LIN {X 0,Y 412.473,Z 356.373,A -85,B 0,C 180,E1 -10488.564,E2 -10488.564} C_VEL
LIN {X 0,Y 413.855,Z 363.338,A -85,B 0,C 180,E1 -10491.872,E2 -10491.872} C_VEL
LIN {X 0,Y 414.561,Z 368.323,A -85,B 0,C 180,E1 -10494.091,E2 -10494.091} C_VEL
LIN {X 0,Y 414.047,Z 374.671,A -85,B 0,C 180,E1 -10496.674,E2 -10496.674} C_VEL
LIN {X 0,Y 413.079,Z 384.313,A -85,B 0,C 180,E1 -10500.435,E2 -10500.435} C_VEL
LIN {X 0,Y 412.15,Z 394.191,A -85,B 0,C 180,E1 -10504.226,E2 -10504.226} C_VEL
LIN {X 0,Y 411.927,Z 397.665,A -85,B 0,C 180,E1 -10505.56,E2 -10505.56} C_VEL
LIN {X 0,Y 415.986,Z 414.745,A -85,B 0,C 180,E1 -10506.23,E2 -10506.23} C_VEL
LIN {X 0,Y 418.674,Z 429.42,A -85,B 0,C 180,E1 -10506.952,E2 -10506.952} C_VEL
LIN {X 0,Y 419.189,Z 434.682,A -85,B 0,C 180,E1 -10507.237,E2 -10507.237} C_VEL
LIN {X 0,Y 418.226,Z 448.445,A -85,B 0,C 180,E1 -10507.985,E2 -10507.985} C_VEL
LIN {X 0,Y 417.116,Z 461.685,A -85,B 0,C 180,E1 -10508.89,E2 -10508.89} C_VEL
LIN {X 0,Y 415.821,Z 474.731,A -85,B 0,C 180,E1 -10509.985,E2 -10509.985} C_VEL
LIN {X 0,Y 414.639,Z 486.804,A -85,B 0,C 180,E1 -10511.213,E2 -10511.213} C_VEL
LIN {X 0,Y 413.542,Z 498.914,A -85,B 0,C 180,E1 -10512.698,E2 -10512.698} C_VEL
LIN {X 0,Y 412.48,Z 509.113,A -85,B 0,C 180,E1 -10514.18,E2 -10514.18} C_VEL
LIN {X 0,Y 411.633,Z 519.099,A -85,B 0,C 180,E1 -10515.919,E2 -10515.919} C_VEL
LIN {X 0,Y 410.992,Z 527.441,A -85,B 0,C 180,E1 -10517.658,E2 -10517.658} C_VEL
LIN {X 0,Y 410.621,Z 533.414,A -85,B 0,C 180,E1 -10519.148,E2 -10519.148} C_VEL
LIN {X 0,Y 410.225,Z 539.99,A -85,B 0,C 180,E1 -10521.13,E2 -10521.13} C_VEL
LIN {X 0,Y 410.058,Z 545.099,A -85,B 0,C 180,E1 -10523.109,E2 -10523.109} C_VEL
LIN {X 0,Y 409.992,Z 548.857,A -85,B 0,C 180,E1 -10525.083,E2 -10525.083} C_VEL
LIN {X 0,Y 409.971,Z 551.337,A -85,B 0,C 180,E1 -10527.052,E2 -10527.052} C_VEL
LIN {X 0,Y 409.974,Z 552.586,A -85,B 0,C 180,E1 -10529.018,E2 -10529.018} C_VEL
LIN {X 0,Y 409.974,Z 552.585,A -85,B 0,C 180,E1 -10530.982,E2 -10530.982} C_VEL
LIN {X 0,Y 409.971,Z 551.33,A -85,B 0,C 180,E1 -10532.948,E2 -10532.948} C_VEL
LIN {X 0,Y 409.998,Z 548.848,A -85,B 0,C 180,E1 -10534.917,E2 -10534.917} C_VEL
LIN {X 0,Y 410.068,Z 545.095,A -85,B 0,C 180,E1 -10536.89,E2 -10536.89} C_VEL
LIN {X 0,Y 410.225,Z 539.984,A -85,B 0,C 180,E1 -10538.87,E2 -10538.87} C_VEL
LIN {X 0,Y 410.621,Z 533.397,A -85,B 0,C 180,E1 -10540.852,E2 -10540.852} C_VEL
LIN {X 0,Y 411.011,Z 526.298,A -85,B 0,C 180,E1 -10542.593,E2 -10542.593} C_VEL
LIN {X 0,Y 411.745,Z 517.767,A -85,B 0,C 180,E1 -10544.33,E2 -10544.33} C_VEL
LIN {X 0,Y 412.642,Z 507.498,A -85,B 0,C 180,E1 -10546.067,E2 -10546.067} C_VEL
LIN {X 0,Y 413.651,Z 497.039,A -85,B 0,C 180,E1 -10547.552,E2 -10547.552} C_VEL
LIN {X 0,Y 414.933,Z 484.534,A -85,B 0,C 180,E1 -10549.029,E2 -10549.029} C_VEL
LIN {X 0,Y 416.072,Z 472.024,A -85,B 0,C 180,E1 -10550.26,E2 -10550.26} C_VEL
LIN {X 0,Y 417.353,Z 458.355,A -85,B 0,C 180,E1 -10551.356,E2 -10551.356} C_VEL
LIN {X 0,Y 418.476,Z 445.087,A -85,B 0,C 180,E1 -10552.215,E2 -10552.215} C_VEL
LIN {X 0,Y 419.176,Z 432.684,A -85,B 0,C 180,E1 -10552.861,E2 -10552.861} C_VEL
LIN {X 0,Y 416.901,Z 419.271,A -85,B 0,C 180,E1 -10553.554,E2 -10553.554} C_VEL
LIN {X 0,Y 413.581,Z 404.549,A -85,B 0,C 180,E1 -10554.182,E2 -10554.182} C_VEL
LIN {X 0,Y 411.925,Z 397.627,A -85,B 0,C 180,E1 -10554.44,E2 -10554.44} C_VEL
LIN {X 0,Y 412.667,Z 388.34,A -85,B 0,C 180,E1 -10558.01,E2 -10558.01} C_VEL
LIN {X 0,Y 413.477,Z 380.023,A -85,B 0,C 180,E1 -10561.226,E2 -10561.226} C_VEL
LIN {X 0,Y 414.356,Z 371.385,A -85,B 0,C 180,E1 -10564.625,E2 -10564.625} C_VEL
LIN {X 0,Y 414.582,Z 368.286,A -85,B 0,C 180,E1 -10565.908,E2 -10565.908} C_VEL
LIN {X 0,Y 413.649,Z 362.257,A -85,B 0,C 180,E1 -10568.597,E2 -10568.597} C_VEL
LIN {X 0,Y 412.154,Z 354.701,A -85,B 0,C 180,E1 -10572.237,E2 -10572.237} C_VEL
LIN {X 0,Y 411.206,Z 349.895,A -85,B 0,C 180,E1 -10574.733,E2 -10574.733} C_VEL
LIN {X 0,Y 411.2,Z 349.883,A -85,B 0,C 180,E1 -10578.198,E2 -10578.198} C_VEL
LIN {X 0,Y 411.234,Z 349.887,A -85,B 0,C 180,E1 -10580.778,E2 -10580.778} C_VEL
LIN {X 0,Y 411.202,Z 349.895,A -85,B 0,C 180,E1 -10584.472,E2 -10584.472} C_VEL
LIN {X 0,Y 411.209,Z 349.892,A -85,B 0,C 180,E1 -10586.874,E2 -10586.874} C_VEL
LIN {X 0,Y 411.235,Z 349.886,A -85,B 0,C 180,E1 -10590.644,E2 -10590.644} C_VEL
LIN {X 0,Y 411.241,Z 349.885,A -85,B 0,C 180,E1 -10593.619,E2 -10593.619} C_VEL
LIN {X 0,Y 411.207,Z 349.888,A -85,B 0,C 180,E1 -10596.853,E2 -10596.853} C_VEL
LIN {X 0,Y 411.219,Z 349.887,A -85,B 0,C 180,E1 -10600.05,E2 -10600.05} C_VEL
LIN {X 0,Y 411.266,Z 349.881,A -85,B 0,C 180,E1 -10603.131,E2 -10603.131} C_VEL
LIN {X 0,Y 411.317,Z 349.87,A -85,B 0,C 180,E1 -10606.891,E2 -10606.891} C_VEL
LIN {X 0,Y 411.298,Z 349.874,A -85,B 0,C 180,E1 -10610.162,E2 -10610.162} C_VEL
LIN {X 0,Y 411.447,Z 349.857,A -85,B 0,C 180,E1 -10613.133,E2 -10613.133} C_VEL
LIN {X 0,Y 411.313,Z 349.877,A -85,B 0,C 180,E1 -10615.099,E2 -10615.099} C_VEL
LIN {X 0,Y 411.516,Z 349.849,A -85,B 0,C 180,E1 -10618.043,E2 -10618.043} C_VEL
LIN {X 0,Y 411.645,Z 349.831,A -85,B 0,C 180,E1 -10620,E2 -10620} C_VEL
LIN {X 0,Y 411.461,Z 349.858,A -85,B 0,C 180,E1 -10622.937,E2 -10622.937} C_VEL
LIN {X 0,Y 411.465,Z 349.855,A -85,B 0,C 180,E1 -10626.867,E2 -10626.867} C_VEL
LIN {X 0,Y 411.311,Z 349.878,A -85,B 0,C 180,E1 -10629.838,E2 -10629.838} C_VEL
LIN {X 0,Y 411.318,Z 349.876,A -85,B 0,C 180,E1 -10633.109,E2 -10633.109} C_VEL
LIN {X 0,Y 411.261,Z 349.882,A -85,B 0,C 180,E1 -10636.889,E2 -10636.889} C_VEL
LIN {X 0,Y 411.234,Z 349.888,A -85,B 0,C 180,E1 -10639.987,E2 -10639.987} C_VEL
LIN {X 0,Y 411.207,Z 349.89,A -85,B 0,C 180,E1 -10643.147,E2 -10643.147} C_VEL
LIN {X 0,Y 411.242,Z 349.884,A -85,B 0,C 180,E1 -10646.381,E2 -10646.381} C_VEL
LIN {X 0,Y 411.204,Z 349.886,A -85,B 0,C 180,E1 -10649.713,E2 -10649.713} C_VEL
LIN {X 0,Y 411.21,Z 349.888,A -85,B 0,C 180,E1 -10653.156,E2 -10653.156} C_VEL
LIN {X 0,Y 411.196,Z 349.891,A -85,B 0,C 180,E1 -10656.553,E2 -10656.553} C_VEL
LIN {X 0,Y 411.216,Z 349.889,A -85,B 0,C 180,E1 -10659.728,E2 -10659.728} C_VEL
LIN {X 0,Y 411.177,Z 349.893,A -85,B 0,C 180,E1 -10663.133,E2 -10663.133} C_VEL
LIN {X 0,Y 411.171,Z 349.896,A -85,B 0,C 180,E1 -10665.881,E2 -10665.881} C_VEL
LIN {X 0,Y 411.242,Z 350.049,A -85,B 0,C 180,E1 -10667.531,E2 -10667.531} C_VEL
LIN {X 0,Y 411.73,Z 353.5,A -85,B 0,C 180,E1 -10670.186,E2 -10670.186} C_VEL
LIN {X 0,Y 411.809,Z 356.083,A -85,B 0,C 180,E1 -10672.093,E2 -10672.093} C_VEL
LIN {X 0,Y 411.664,Z 360.213,A -85,B 0,C 180,E1 -10675.032,E2 -10675.032} C_VEL
LIN {X 0,Y 411.374,Z 364.529,A -85,B 0,C 180,E1 -10678.021,E2 -10678.021} C_VEL
LIN {X 0,Y 411.101,Z 369.543,A -85,B 0,C 180,E1 -10681.401,E2 -10681.401} C_VEL
LIN {X 0,Y 410.923,Z 374.622,A -85,B 0,C 180,E1 -10684.686,E2 -10684.686} C_VEL
LIN {X 0,Y 410.712,Z 380.389,A -85,B 0,C 180,E1 -10688.235,E2 -10688.235} C_VEL
LIN {X 0,Y 415.732,Z 397.121,A -85,B 0,C 180,E1 -10688.991,E2 -10688.991} C_VEL
LIN {X 0,Y 418.903,Z 410.203,A -85,B 0,C 180,E1 -10689.72,E2 -10689.72} C_VEL
LIN {X 0,Y 418.637,Z 418.558,A -85,B 0,C 180,E1 -10690.151,E2 -10690.151} C_VEL
LIN {X 0,Y 417.778,Z 431.637,A -85,B 0,C 180,E1 -10690.978,E2 -10690.978} C_VEL
LIN {X 0,Y 416.805,Z 443.798,A -85,B 0,C 180,E1 -10691.951,E2 -10691.951} C_VEL
LIN {X 0,Y 415.674,Z 454.932,A -85,B 0,C 180,E1 -10693.043,E2 -10693.043} C_VEL
LIN {X 0,Y 414.628,Z 465.155,A -85,B 0,C 180,E1 -10694.264,E2 -10694.264} C_VEL
LIN {X 0,Y 413.718,Z 473.99,A -85,B 0,C 180,E1 -10695.532,E2 -10695.532} C_VEL
LIN {X 0,Y 412.839,Z 482.36,A -85,B 0,C 180,E1 -10696.964,E2 -10696.964} C_VEL
LIN {X 0,Y 411.999,Z 489.544,A -85,B 0,C 180,E1 -10698.438,E2 -10698.438} C_VEL
LIN {X 0,Y 411.306,Z 496.408,A -85,B 0,C 180,E1 -10700.162,E2 -10700.162} C_VEL
LIN {X 0,Y 410.725,Z 502.566,A -85,B 0,C 180,E1 -10702.132,E2 -10702.132} C_VEL
LIN {X 0,Y 410.437,Z 507.144,A -85,B 0,C 180,E1 -10704.103,E2 -10704.103} C_VEL
LIN {X 0,Y 410.166,Z 510.317,A -85,B 0,C 180,E1 -10706.07,E2 -10706.07} C_VEL
LIN {X 0,Y 410.071,Z 512.187,A -85,B 0,C 180,E1 -10708.036,E2 -10708.036} C_VEL
LIN {X 0,Y 409.971,Z 512.826,A -85,B 0,C 180,E1 -10710,E2 -10710} C_VEL
LIN {X 0,Y 410.07,Z 512.25,A -85,B 0,C 180,E1 -10711.964,E2 -10711.964} C_VEL
LIN {X 0,Y 410.164,Z 510.414,A -85,B 0,C 180,E1 -10713.954,E2 -10713.954} C_VEL
LIN {X 0,Y 410.432,Z 507.339,A -85,B 0,C 180,E1 -10715.897,E2 -10715.897} C_VEL
LIN {X 0,Y 410.722,Z 502.824,A -85,B 0,C 180,E1 -10717.868,E2 -10717.868} C_VEL
LIN {X 0,Y 410.764,Z 502.241,A -85,B 0,C 180,E1 -10718.078,E2 -10718.078} C_VEL
LIN {X 0,Y 410.259,Z 500.112,A -85,B 0,C 180,E1 -10718.844,E2 -10718.844} C_VEL
LIN {X 0,Y 407.69,Z 496.379,A -85,B 0,C 180,E1 -10720.086,E2 -10720.086} C_VEL
LIN {X 0,Y 405.311,Z 492.191,A -85,B 0,C 180,E1 -10721.307,E2 -10721.307} C_VEL
LIN {X 0,Y 405.102,Z 489.194,A -85,B 0,C 180,E1 -10722.029,E2 -10722.029} C_VEL
LIN {X 0,Y 406.031,Z 481.921,A -85,B 0,C 180,E1 -10723.514,E2 -10723.514} C_VEL
LIN {X 0,Y 406.961,Z 473.123,A -85,B 0,C 180,E1 -10725.013,E2 -10725.013} C_VEL
LIN {X 0,Y 407.969,Z 464.366,A -85,B 0,C 180,E1 -10726.257,E2 -10726.257} C_VEL
LIN {X 0,Y 409.145,Z 452.742,A -85,B 0,C 180,E1 -10727.623,E2 -10727.623} C_VEL
LIN {X 0,Y 410.309,Z 441.068,A -85,B 0,C 180,E1 -10728.733,E2 -10728.733} C_VEL
LIN {X 0,Y 411.399,Z 428.167,A -85,B 0,C 180,E1 -10729.718,E2 -10729.718} C_VEL
LIN {X 0,Y 412.277,Z 415.028,A -85,B 0,C 180,E1 -10730.501,E2 -10730.501} C_VEL
LIN {X 0,Y 412.268,Z 411.549,A -85,B 0,C 180,E1 -10730.687,E2 -10730.687} C_VEL
LIN {X 0,Y 409.079,Z 398.314,A -85,B 0,C 180,E1 -10731.455,E2 -10731.455} C_VEL
LIN {X 0,Y 404.658,Z 383.818,A -85,B 0,C 180,E1 -10732.15,E2 -10732.15} C_VEL
LIN {X 0,Y 403.732,Z 380.544,A -85,B 0,C 180,E1 -10732.295,E2 -10732.295} C_VEL
LIN {X 0,Y 403.891,Z 374.995,A -85,B 0,C 180,E1 -10735.787,E2 -10735.787} C_VEL
LIN {X 0,Y 404.125,Z 369.877,A -85,B 0,C 180,E1 -10739.14,E2 -10739.14} C_VEL
LIN {X 0,Y 404.396,Z 364.864,A -85,B 0,C 180,E1 -10742.599,E2 -10742.599} C_VEL
LIN {X 0,Y 404.7,Z 359.772,A -85,B 0,C 180,E1 -10746.189,E2 -10746.189} C_VEL
LIN {X 0,Y 404.856,Z 356.353,A -85,B 0,C 180,E1 -10748.678,E2 -10748.678} C_VEL
LIN {X 0,Y 404.475,Z 352.452,A -85,B 0,C 180,E1 -10751.656,E2 -10751.656} C_VEL
LIN {X 0,Y 404.18,Z 350.766,A -85,B 0,C 180,E1 -10753.087,E2 -10753.087} C_VEL
LIN {X 0,Y 404.157,Z 350.765,A -85,B 0,C 180,E1 -10756.916,E2 -10756.916} C_VEL
LIN {X 0,Y 404.173,Z 350.763,A -85,B 0,C 180,E1 -10759.956,E2 -10759.956} C_VEL
LIN {X 0,Y 404.141,Z 350.77,A -85,B 0,C 180,E1 -10763.125,E2 -10763.125} C_VEL
LIN {X 0,Y 404.149,Z 350.767,A -85,B 0,C 180,E1 -10766.188,E2 -10766.188} C_VEL
LIN {X 0,Y 404.15,Z 350.768,A -85,B 0,C 180,E1 -10769.715,E2 -10769.715} C_VEL
LIN {X 0,Y 404.201,Z 350.764,A -85,B 0,C 180,E1 -10773.123,E2 -10773.123} C_VEL
LIN {X 0,Y 404.182,Z 350.764,A -85,B 0,C 180,E1 -10775.334,E2 -10775.334} C_VEL
LIN {X 0,Y 404.144,Z 350.766,A -85,B 0,C 180,E1 -10778.581,E2 -10778.581} C_VEL
LIN {X 0,Y 404.214,Z 350.758,A -85,B 0,C 180,E1 -10781.762,E2 -10781.762} C_VEL
LIN {X 0,Y 404.212,Z 350.758,A -85,B 0,C 180,E1 -10784.882,E2 -10784.882} C_VEL
LIN {X 0,Y 404.262,Z 350.752,A -85,B 0,C 180,E1 -10787.958,E2 -10787.958} C_VEL
LIN {X 0,Y 404.439,Z 350.732,A -85,B 0,C 180,E1 -10792.099,E2 -10792.099} C_VEL
LIN {X 0,Y 404.43,Z 350.73,A -85,B 0,C 180,E1 -10794.015,E2 -10794.015} C_VEL
LIN {X 0,Y 404.486,Z 350.723,A -85,B 0,C 180,E1 -10798.008,E2 -10798.008} C_VEL
LIN {X 0,Y 404.615,Z 350.712,A -85,B 0,C 180,E1 -10800,E2 -10800} C_VEL
LIN {X 0,Y 404.42,Z 350.733,A -85,B 0,C 180,E1 -10802.988,E2 -10802.988} C_VEL
LIN {X 0,Y 404.419,Z 350.733,A -85,B 0,C 180,E1 -10805.985,E2 -10805.985} C_VEL
LIN {X 0,Y 404.272,Z 350.754,A -85,B 0,C 180,E1 -10809.001,E2 -10809.001} C_VEL
LIN {X 0,Y 404.274,Z 350.756,A -85,B 0,C 180,E1 -10812.041,E2 -10812.041} C_VEL
LIN {X 0,Y 404.213,Z 350.763,A -85,B 0,C 180,E1 -10815.118,E2 -10815.118} C_VEL
LIN {X 0,Y 404.215,Z 350.763,A -85,B 0,C 180,E1 -10818.238,E2 -10818.238} C_VEL
LIN {X 0,Y 404.144,Z 350.771,A -85,B 0,C 180,E1 -10821.419,E2 -10821.419} C_VEL
LIN {X 0,Y 404.181,Z 350.764,A -85,B 0,C 180,E1 -10824.665,E2 -10824.665} C_VEL
LIN {X 0,Y 404.199,Z 350.761,A -85,B 0,C 180,E1 -10827.999,E2 -10827.999} C_VEL
LIN {X 0,Y 404.143,Z 350.771,A -85,B 0,C 180,E1 -10831.558,E2 -10831.558} C_VEL
LIN {X 0,Y 404.189,Z 350.766,A -85,B 0,C 180,E1 -10835.016,E2 -10835.016} C_VEL
LIN {X 0,Y 404.159,Z 350.769,A -85,B 0,C 180,E1 -10838.756,E2 -10838.756} C_VEL
LIN {X 0,Y 404.125,Z 350.772,A -85,B 0,C 180,E1 -10841.599,E2 -10841.599} C_VEL
LIN {X 0,Y 404.167,Z 350.933,A -85,B 0,C 180,E1 -10844.823,E2 -10844.823} C_VEL
LIN {X 0,Y 405.185,Z 355.851,A -85,B 0,C 180,E1 -10847.432,E2 -10847.432} C_VEL
LIN {X 0,Y 406.58,Z 363.235,A -85,B 0,C 180,E1 -10851.064,E2 -10851.064} C_VEL
LIN {X 0,Y 407.518,Z 368.477,A -85,B 0,C 180,E1 -10853.488,E2 -10853.488} C_VEL
LIN {X 0,Y 407.416,Z 372.727,A -85,B 0,C 180,E1 -10855.301,E2 -10855.301} C_VEL
LIN {X 0,Y 406.602,Z 380.162,A -85,B 0,C 180,E1 -10858.309,E2 -10858.309} C_VEL
LIN {X 0,Y 405.746,Z 388.353,A -85,B 0,C 180,E1 -10861.554,E2 -10861.554} C_VEL
LIN {X 0,Y 404.933,Z 397.498,A -85,B 0,C 180,E1 -10865.141,E2 -10865.141} C_VEL
LIN {X 0,Y 409.001,Z 414.267,A -85,B 0,C 180,E1 -10865.816,E2 -10865.816} C_VEL
LIN {X 0,Y 411.843,Z 429.09,A -85,B 0,C 180,E1 -10866.568,E2 -10866.568} C_VEL
LIN {X 0,Y 412.502,Z 435.595,A -85,B 0,C 180,E1 -10866.929,E2 -10866.929} C_VEL
LIN {X 0,Y 411.441,Z 449.77,A -85,B 0,C 180,E1 -10867.73,E2 -10867.73} C_VEL
LIN {X 0,Y 410.13,Z 464.317,A -85,B 0,C 180,E1 -10868.777,E2 -10868.777} C_VEL
LIN {X 0,Y 408.883,Z 476.849,A -85,B 0,C 180,E1 -10869.893,E2 -10869.893} C_VEL
LIN {X 0,Y 407.57,Z 489.439,A -85,B 0,C 180,E1 -10871.247,E2 -10871.247} C_VEL
LIN {X 0,Y 406.489,Z 500.302,A -85,B 0,C 180,E1 -10872.648,E2 -10872.648} C_VEL
LIN {X 0,Y 405.437,Z 510.226,A -85,B 0,C 180,E1 -10874.156,E2 -10874.156} C_VEL
LIN {X 0,Y 404.552,Z 519.973,A -85,B 0,C 180,E1 -10875.924,E2 -10875.924} C_VEL
LIN {X 0,Y 403.897,Z 528.103,A -85,B 0,C 180,E1 -10877.692,E2 -10877.692} C_VEL
LIN {X 0,Y 403.418,Z 534.859,A -85,B 0,C 180,E1 -10879.46,E2 -10879.46} C_VEL
LIN {X 0,Y 403.114,Z 541.068,A -85,B 0,C 180,E1 -10881.478,E2 -10881.478} C_VEL
LIN {X 0,Y 402.982,Z 544.744,A -85,B 0,C 180,E1 -10882.988,E2 -10882.988} C_VEL
LIN {X 0,Y 402.902,Z 548.506,A -85,B 0,C 180,E1 -10884.996,E2 -10884.996} C_VEL
LIN {X 0,Y 402.872,Z 550.989,A -85,B 0,C 180,E1 -10887,E2 -10887} C_VEL
LIN {X 0,Y 402.899,Z 552.241,A -85,B 0,C 180,E1 -10889,E2 -10889} C_VEL
LIN {X 0,Y 402.899,Z 552.24,A -85,B 0,C 180,E1 -10890.999,E2 -10890.999} C_VEL
LIN {X 0,Y 402.872,Z 550.982,A -85,B 0,C 180,E1 -10893,E2 -10893} C_VEL
LIN {X 0,Y 402.912,Z 548.497,A -85,B 0,C 180,E1 -10895.003,E2 -10895.003} C_VEL
LIN {X 0,Y 402.989,Z 544.738,A -85,B 0,C 180,E1 -10897.012,E2 -10897.012} C_VEL
LIN {X 0,Y 403.149,Z 539.619,A -85,B 0,C 180,E1 -10899.027,E2 -10899.027} C_VEL
LIN {X 0,Y 403.572,Z 533.024,A -85,B 0,C 180,E1 -10901.044,E2 -10901.044} C_VEL
LIN {X 0,Y 404.072,Z 524.767,A -85,B 0,C 180,E1 -10903.068,E2 -10903.068} C_VEL
LIN {X 0,Y 404.89,Z 515.987,A -85,B 0,C 180,E1 -10904.835,E2 -10904.835} C_VEL
LIN {X 0,Y 405.919,Z 505.434,A -85,B 0,C 180,E1 -10906.599,E2 -10906.599} C_VEL
LIN {X 0,Y 407.142,Z 493.616,A -85,B 0,C 180,E1 -10908.237,E2 -10908.237} C_VEL
LIN {X 0,Y 408.323,Z 481.713,A -85,B 0,C 180,E1 -10909.611,E2 -10909.611} C_VEL
LIN {X 0,Y 409.655,Z 468.681,A -85,B 0,C 180,E1 -10910.854,E2 -10910.854} C_VEL
LIN {X 0,Y 410.848,Z 456.055,A -85,B 0,C 180,E1 -10911.843,E2 -10911.843} C_VEL
LIN {X 0,Y 412.031,Z 441.745,A -85,B 0,C 180,E1 -10912.744,E2 -10912.744} C_VEL
LIN {X 0,Y 412.538,Z 434.213,A -85,B 0,C 180,E1 -10913.135,E2 -10913.135} C_VEL
LIN {X 0,Y 410.302,Z 420.672,A -85,B 0,C 180,E1 -10913.871,E2 -10913.871} C_VEL
LIN {X 0,Y 407.141,Z 406.39,A -85,B 0,C 180,E1 -10914.516,E2 -10914.516} C_VEL
LIN {X 0,Y 404.958,Z 397.41,A -85,B 0,C 180,E1 -10914.882,E2 -10914.882} C_VEL
LIN {X 0,Y 405.752,Z 388.345,A -85,B 0,C 180,E1 -10918.445,E2 -10918.445} C_VEL
LIN {X 0,Y 406.697,Z 379.029,A -85,B 0,C 180,E1 -10922.14,E2 -10922.14} C_VEL
LIN {X 0,Y 407.585,Z 371.277,A -85,B 0,C 180,E1 -10925.276,E2 -10925.276} C_VEL
LIN {X 0,Y 407.307,Z 367.001,A -85,B 0,C 180,E1 -10927.151,E2 -10927.151} C_VEL
LIN {X 0,Y 405.984,Z 360.177,A -85,B 0,C 180,E1 -10930.387,E2 -10930.387} C_VEL
LIN {X 0,Y 404.928,Z 354.602,A -85,B 0,C 180,E1 -10933.201,E2 -10933.201} C_VEL
LIN {X 0,Y 404.135,Z 350.768,A -85,B 0,C 180,E1 -10935.303,E2 -10935.303} C_VEL
LIN {X 0,Y 404.153,Z 350.758,A -85,B 0,C 180,E1 -10938.639,E2 -10938.639} C_VEL
LIN {X 0,Y 404.164,Z 350.769,A -85,B 0,C 180,E1 -10941.491,E2 -10941.491} C_VEL
LIN {X 0,Y 404.188,Z 350.768,A -85,B 0,C 180,E1 -10944.984,E2 -10944.984} C_VEL
LIN {X 0,Y 404.144,Z 350.771,A -85,B 0,C 180,E1 -10948.554,E2 -10948.554} C_VEL
LIN {X 0,Y 404.198,Z 350.761,A -85,B 0,C 180,E1 -10952.001,E2 -10952.001} C_VEL
LIN {X 0,Y 404.18,Z 350.764,A -85,B 0,C 180,E1 -10955.335,E2 -10955.335} C_VEL
LIN {X 0,Y 404.142,Z 350.764,A -85,B 0,C 180,E1 -10958.581,E2 -10958.581} C_VEL
LIN {X 0,Y 404.214,Z 350.758,A -85,B 0,C 180,E1 -10961.762,E2 -10961.762} C_VEL
LIN {X 0,Y 404.212,Z 350.759,A -85,B 0,C 180,E1 -10964.882,E2 -10964.882} C_VEL
LIN {X 0,Y 404.273,Z 350.75,A -85,B 0,C 180,E1 -10967.959,E2 -10967.959} C_VEL
LIN {X 0,Y 404.27,Z 350.749,A -85,B 0,C 180,E1 -10970.999,E2 -10970.999} C_VEL
LIN {X 0,Y 404.422,Z 350.729,A -85,B 0,C 180,E1 -10974.015,E2 -10974.015} C_VEL
LIN {X 0,Y 404.484,Z 350.724,A -85,B 0,C 180,E1 -10978.009,E2 -10978.009} C_VEL
LIN {X 0,Y 404.614,Z 350.707,A -85,B 0,C 180,E1 -10980,E2 -10980} C_VEL
LIN {X 0,Y 404.42,Z 350.736,A -85,B 0,C 180,E1 -10982.989,E2 -10982.989} C_VEL
LIN {X 0,Y 404.416,Z 350.732,A -85,B 0,C 180,E1 -10986.987,E2 -10986.987} C_VEL
LIN {X 0,Y 404.274,Z 350.754,A -85,B 0,C 180,E1 -10990.011,E2 -10990.011} C_VEL
LIN {X 0,Y 404.27,Z 350.755,A -85,B 0,C 180,E1 -10993.211,E2 -10993.211} C_VEL
LIN {X 0,Y 404.22,Z 350.758,A -85,B 0,C 180,E1 -10997.007,E2 -10997.007} C_VEL
LIN {X 0,Y 404.168,Z 350.764,A -85,B 0,C 180,E1 -11000.352,E2 -11000.352} C_VEL
LIN {X 0,Y 404.173,Z 350.763,A -85,B 0,C 180,E1 -11003.574,E2 -11003.574} C_VEL
LIN {X 0,Y 404.187,Z 350.762,A -85,B 0,C 180,E1 -11005.766,E2 -11005.766} C_VEL
LIN {X 0,Y 404.199,Z 350.76,A -85,B 0,C 180,E1 -11008,E2 -11008} C_VEL
LIN {X 0,Y 404.143,Z 350.769,A -85,B 0,C 180,E1 -11011.558,E2 -11011.558} C_VEL
LIN {X 0,Y 404.188,Z 350.765,A -85,B 0,C 180,E1 -11015.016,E2 -11015.016} C_VEL
LIN {X 0,Y 404.157,Z 350.768,A -85,B 0,C 180,E1 -11018.757,E2 -11018.757} C_VEL
LIN {X 0,Y 404.126,Z 350.772,A -85,B 0,C 180,E1 -11021.6,E2 -11021.6} C_VEL
LIN {X 0,Y 404.148,Z 350.77,A -85,B 0,C 180,E1 -11024.522,E2 -11024.522} C_VEL
LIN {X 0,Y 404.165,Z 350.775,A -85,B 0,C 180,E1 -11027.107,E2 -11027.107} C_VEL
LIN {X 0,Y 404.706,Z 354.472,A -85,B 0,C 180,E1 -11030.019,E2 -11030.019} C_VEL
LIN {X 0,Y 404.769,Z 357.892,A -85,B 0,C 180,E1 -11032.576,E2 -11032.576} C_VEL
LIN {X 0,Y 404.64,Z 361.299,A -85,B 0,C 180,E1 -11035.029,E2 -11035.029} C_VEL
LIN {X 0,Y 404.336,Z 366.351,A -85,B 0,C 180,E1 -11038.57,E2 -11038.57} C_VEL
LIN {X 0,Y 404.025,Z 371.415,A -85,B 0,C 180,E1 -11041.987,E2 -11041.987} C_VEL
LIN {X 0,Y 403.832,Z 376.534,A -85,B 0,C 180,E1 -11045.312,E2 -11045.312} C_VEL
LIN {X 0,Y 403.72,Z 380.559,A -85,B 0,C 180,E1 -11047.809,E2 -11047.809} C_VEL
LIN {X 0,Y 408.667,Z 396.984,A -85,B 0,C 180,E1 -11048.571,E2 -11048.571} C_VEL
LIN {X 0,Y 411.894,Z 409.71,A -85,B 0,C 180,E1 -11049.298,E2 -11049.298} C_VEL
LIN {X 0,Y 412.43,Z 412.885,A -85,B 0,C 180,E1 -11049.485,E2 -11049.485} C_VEL
LIN {X 0,Y 411.64,Z 424.913,A -85,B 0,C 180,E1 -11050.164,E2 -11050.164} C_VEL
LIN {X 0,Y 410.629,Z 436.995,A -85,B 0,C 180,E1 -11051.023,E2 -11051.023} C_VEL
LIN {X 0,Y 409.648,Z 448.183,A -85,B 0,C 180,E1 -11052.012,E2 -11052.012} C_VEL
LIN {X 0,Y 408.469,Z 459.659,A -85,B 0,C 180,E1 -11053.25,E2 -11053.25} C_VEL
LIN {X 0,Y 407.404,Z 469.148,A -85,B 0,C 180,E1 -11054.491,E2 -11054.491} C_VEL
LIN {X 0,Y 406.359,Z 478.641,A -85,B 0,C 180,E1 -11055.988,E2 -11055.988} C_VEL
LIN {X 0,Y 405.433,Z 486.499,A -85,B 0,C 180,E1 -11057.486,E2 -11057.486} C_VEL
LIN {X 0,Y 404.73,Z 493.043,A -85,B 0,C 180,E1 -11058.988,E2 -11058.988} C_VEL
LIN {X 0,Y 404.153,Z 498.499,A -85,B 0,C 180,E1 -11060.491,E2 -11060.491} C_VEL
LIN {X 0,Y 403.601,Z 504.207,A -85,B 0,C 180,E1 -11062.496,E2 -11062.496} C_VEL
LIN {X 0,Y 403.39,Z 507.497,A -85,B 0,C 180,E1 -11064,E2 -11064} C_VEL
LIN {X 0,Y 403.08,Z 510.667,A -85,B 0,C 180,E1 -11066.001,E2 -11066.001} C_VEL
LIN {X 0,Y 403.002,Z 512.533,A -85,B 0,C 180,E1 -11068.001,E2 -11068.001} C_VEL
LIN {X 0,Y 402.894,Z 513.171,A -85,B 0,C 180,E1 -11070,E2 -11070} C_VEL
LIN {X 0,Y 403.002,Z 512.594,A -85,B 0,C 180,E1 -11071.999,E2 -11071.999} C_VEL
LIN {X 0,Y 403.079,Z 510.795,A -85,B 0,C 180,E1 -11073.999,E2 -11073.999} C_VEL
LIN {X 0,Y 403.386,Z 507.689,A -85,B 0,C 180,E1 -11076.001,E2 -11076.001} C_VEL
LIN {X 0,Y 403.697,Z 503.18,A -85,B 0,C 180,E1 -11078.006,E2 -11078.006} C_VEL
LIN {X 0,Y 404.26,Z 497.11,A -85,B 0,C 180,E1 -11080.012,E2 -11080.012} C_VEL
LIN {X 0,Y 404.992,Z 490.335,A -85,B 0,C 180,E1 -11081.765,E2 -11081.765} C_VEL
LIN {X 0,Y 405.102,Z 489.194,A -85,B 0,C 180,E1 -11082.029,E2 -11082.029} C_VEL
LIN {X 0,Y 404.931,Z 486.066,A -85,B 0,C 180,E1 -11082.737,E2 -11082.737} C_VEL
LIN {X 0,Y 402.774,Z 480.812,A -85,B 0,C 180,E1 -11083.893,E2 -11083.893} C_VEL
LIN {X 0,Y 400.585,Z 475.063,A -85,B 0,C 180,E1 -11085.009,E2 -11085.009} C_VEL
LIN {X 0,Y 400.364,Z 471.155,A -85,B 0,C 180,E1 -11085.645,E2 -11085.645} C_VEL
LIN {X 0,Y 401.641,Z 460.876,A -85,B 0,C 180,E1 -11087.044,E2 -11087.044} C_VEL
LIN {X 0,Y 402.876,Z 449.597,A -85,B 0,C 180,E1 -11088.301,E2 -11088.301} C_VEL
LIN {X 0,Y 404.118,Z 437.098,A -85,B 0,C 180,E1 -11089.426,E2 -11089.426} C_VEL
LIN {X 0,Y 405.112,Z 423.773,A -85,B 0,C 180,E1 -11090.381,E2 -11090.381} C_VEL
LIN {X 0,Y 405.73,Z 414.092,A -85,B 0,C 180,E1 -11090.937,E2 -11090.937} C_VEL
LIN {X 0,Y 403.029,Z 401.832,A -85,B 0,C 180,E1 -11091.685,E2 -11091.685} C_VEL
LIN {X 0,Y 398.883,Z 387.74,A -85,B 0,C 180,E1 -11092.421,E2 -11092.421} C_VEL
LIN {X 0,Y 396.67,Z 380.717,A -85,B 0,C 180,E1 -11092.74,E2 -11092.74} C_VEL
LIN {X 0,Y 396.845,Z 376.494,A -85,B 0,C 180,E1 -11095.418,E2 -11095.418} C_VEL
LIN {X 0,Y 397.019,Z 371.77,A -85,B 0,C 180,E1 -11098.552,E2 -11098.552} C_VEL
LIN {X 0,Y 397.242,Z 368.369,A -85,B 0,C 180,E1 -11100.869,E2 -11100.869} C_VEL
LIN {X 0,Y 397.548,Z 363.305,A -85,B 0,C 180,E1 -11104.452,E2 -11104.452} C_VEL
LIN {X 0,Y 397.823,Z 359.324,A -85,B 0,C 180,E1 -11107.347,E2 -11107.347} C_VEL
LIN {X 0,Y 397.773,Z 356.457,A -85,B 0,C 180,E1 -11109.499,E2 -11109.499} C_VEL
LIN {X 0,Y 397.354,Z 352.994,A -85,B 0,C 180,E1 -11112.23,E2 -11112.23} C_VEL
LIN {X 0,Y 397.116,Z 351.646,A -85,B 0,C 180,E1 -11113.481,E2 -11113.481} C_VEL
LIN {X 0,Y 397.106,Z 351.644,A -85,B 0,C 180,E1 -11116.521,E2 -11116.521} C_VEL
LIN {X 0,Y 397.118,Z 351.64,A -85,B 0,C 180,E1 -11120.423,E2 -11120.423} C_VEL
LIN {X 0,Y 397.112,Z 351.644,A -85,B 0,C 180,E1 -11124.266,E2 -11124.266} C_VEL
LIN {X 0,Y 397.119,Z 351.645,A -85,B 0,C 180,E1 -11126.727,E2 -11126.727} C_VEL
LIN {X 0,Y 397.129,Z 351.643,A -85,B 0,C 180,E1 -11130.296,E2 -11130.296} C_VEL
LIN {X 0,Y 397.199,Z 351.633,A -85,B 0,C 180,E1 -11132.61,E2 -11132.61} C_VEL
LIN {X 0,Y 397.138,Z 351.64,A -85,B 0,C 180,E1 -11135.982,E2 -11135.982} C_VEL
LIN {X 0,Y 397.144,Z 351.638,A -85,B 0,C 180,E1 -11139.705,E2 -11139.705} C_VEL
LIN {X 0,Y 397.187,Z 351.633,A -85,B 0,C 180,E1 -11142.845,E2 -11142.845} C_VEL
LIN {X 0,Y 397.234,Z 351.632,A -85,B 0,C 180,E1 -11146.703,E2 -11146.703} C_VEL
LIN {X 0,Y 397.223,Z 351.631,A -85,B 0,C 180,E1 -11149.809,E2 -11149.809} C_VEL
LIN {X 0,Y 397.37,Z 351.611,A -85,B 0,C 180,E1 -11152.888,E2 -11152.888} C_VEL
LIN {X 0,Y 397.26,Z 351.623,A -85,B 0,C 180,E1 -11154.925,E2 -11154.925} C_VEL
LIN {X 0,Y 397.455,Z 351.599,A -85,B 0,C 180,E1 -11157.973,E2 -11157.973} C_VEL
LIN {X 0,Y 397.585,Z 351.587,A -85,B 0,C 180,E1 -11160,E2 -11160} C_VEL
LIN {X 0,Y 397.38,Z 351.611,A -85,B 0,C 180,E1 -11163.041,E2 -11163.041} C_VEL
LIN {X 0,Y 397.37,Z 351.611,A -85,B 0,C 180,E1 -11166.091,E2 -11166.091} C_VEL
LIN {X 0,Y 397.242,Z 351.629,A -85,B 0,C 180,E1 -11169.162,E2 -11169.162} C_VEL
LIN {X 0,Y 397.234,Z 351.633,A -85,B 0,C 180,E1 -11172.257,E2 -11172.257} C_VEL
LIN {X 0,Y 397.185,Z 351.641,A -85,B 0,C 180,E1 -11175.392,E2 -11175.392} C_VEL
LIN {X 0,Y 397.167,Z 351.644,A -85,B 0,C 180,E1 -11178.573,E2 -11178.573} C_VEL
LIN {X 0,Y 397.102,Z 351.65,A -85,B 0,C 180,E1 -11181.818,E2 -11181.818} C_VEL
LIN {X 0,Y 397.161,Z 351.638,A -85,B 0,C 180,E1 -11185.131,E2 -11185.131} C_VEL
LIN {X 0,Y 397.166,Z 351.638,A -85,B 0,C 180,E1 -11187.776,E2 -11187.776} C_VEL
LIN {X 0,Y 397.082,Z 351.65,A -85,B 0,C 180,E1 -11190.882,E2 -11190.882} C_VEL
LIN {X 0,Y 397.129,Z 351.644,A -85,B 0,C 180,E1 -11194.493,E2 -11194.493} C_VEL
LIN {X 0,Y 397.108,Z 351.647,A -85,B 0,C 180,E1 -11198.274,E2 -11198.274} C_VEL
LIN {X 0,Y 397.091,Z 351.648,A -85,B 0,C 180,E1 -11200.908,E2 -11200.908} C_VEL
LIN {X 0,Y 397.121,Z 351.731,A -85,B 0,C 180,E1 -11204.24,E2 -11204.24} C_VEL
LIN {X 0,Y 398.188,Z 356.969,A -85,B 0,C 180,E1 -11207.093,E2 -11207.093} C_VEL
LIN {X 0,Y 399.548,Z 364.135,A -85,B 0,C 180,E1 -11210.71,E2 -11210.71} C_VEL
LIN {X 0,Y 400.571,Z 369.775,A -85,B 0,C 180,E1 -11213.378,E2 -11213.378} C_VEL
LIN {X 0,Y 400.487,Z 373.872,A -85,B 0,C 180,E1 -11215.169,E2 -11215.169} C_VEL
LIN {X 0,Y 399.644,Z 381.112,A -85,B 0,C 180,E1 -11218.158,E2 -11218.158} C_VEL
LIN {X 0,Y 398.703,Z 389.556,A -85,B 0,C 180,E1 -11221.58,E2 -11221.58} C_VEL
LIN {X 0,Y 397.972,Z 397.296,A -85,B 0,C 180,E1 -11224.695,E2 -11224.695} C_VEL
LIN {X 0,Y 402.125,Z 414.311,A -85,B 0,C 180,E1 -11225.41,E2 -11225.41} C_VEL
LIN {X 0,Y 404.956,Z 428.873,A -85,B 0,C 180,E1 -11226.17,E2 -11226.17} C_VEL
LIN {X 0,Y 405.806,Z 434.908,A -85,B 0,C 180,E1 -11226.526,E2 -11226.526} C_VEL
LIN {X 0,Y 404.932,Z 448.179,A -85,B 0,C 180,E1 -11227.283,E2 -11227.283} C_VEL
LIN {X 0,Y 403.619,Z 462.235,A -85,B 0,C 180,E1 -11228.283,E2 -11228.283} C_VEL
LIN {X 0,Y 402.248,Z 475.087,A -85,B 0,C 180,E1 -11229.413,E2 -11229.413} C_VEL
LIN {X 0,Y 400.801,Z 488.081,A -85,B 0,C 180,E1 -11230.805,E2 -11230.805} C_VEL
LIN {X 0,Y 399.636,Z 499.887,A -85,B 0,C 180,E1 -11232.34,E2 -11232.34} C_VEL
LIN {X 0,Y 398.499,Z 509.827,A -85,B 0,C 180,E1 -11233.873,E2 -11233.873} C_VEL
LIN {X 0,Y 397.586,Z 519.589,A -85,B 0,C 180,E1 -11235.672,E2 -11235.672} C_VEL
LIN {X 0,Y 396.909,Z 527.295,A -85,B 0,C 180,E1 -11237.364,E2 -11237.364} C_VEL
LIN {X 0,Y 396.376,Z 534.494,A -85,B 0,C 180,E1 -11239.27,E2 -11239.27} C_VEL
LIN {X 0,Y 396.048,Z 540.71,A -85,B 0,C 180,E1 -11241.324,E2 -11241.324} C_VEL
LIN {X 0,Y 395.905,Z 544.389,A -85,B 0,C 180,E1 -11242.862,E2 -11242.862} C_VEL
LIN {X 0,Y 395.817,Z 548.156,A -85,B 0,C 180,E1 -11244.907,E2 -11244.907} C_VEL
LIN {X 0,Y 395.773,Z 550.642,A -85,B 0,C 180,E1 -11246.946,E2 -11246.946} C_VEL
LIN {X 0,Y 395.867,Z 551.426,A -85,B 0,C 180,E1 -11247.965,E2 -11247.965} C_VEL
LIN {X 0,Y 395.815,Z 552.058,A -85,B 0,C 180,E1 -11250,E2 -11250} C_VEL
LIN {X 0,Y 395.867,Z 551.421,A -85,B 0,C 180,E1 -11252.035,E2 -11252.035} C_VEL
LIN {X 0,Y 395.776,Z 549.545,A -85,B 0,C 180,E1 -11254.073,E2 -11254.073} C_VEL
LIN {X 0,Y 395.896,Z 546.24,A -85,B 0,C 180,E1 -11256.218,E2 -11256.218} C_VEL
LIN {X 0,Y 395.977,Z 541.996,A -85,B 0,C 180,E1 -11258.163,E2 -11258.163} C_VEL
LIN {X 0,Y 396.216,Z 536.145,A -85,B 0,C 180,E1 -11260.217,E2 -11260.217} C_VEL
LIN {X 0,Y 396.699,Z 529.777,A -85,B 0,C 180,E1 -11262.015,E2 -11262.015} C_VEL
LIN {X 0,Y 397.373,Z 522.081,A -85,B 0,C 180,E1 -11263.814,E2 -11263.814} C_VEL
LIN {X 0,Y 398.23,Z 512.818,A -85,B 0,C 180,E1 -11265.613,E2 -11265.613} C_VEL
LIN {X 0,Y 399.398,Z 501.649,A -85,B 0,C 180,E1 -11267.406,E2 -11267.406} C_VEL
LIN {X 0,Y 400.626,Z 490.197,A -85,B 0,C 180,E1 -11268.937,E2 -11268.937} C_VEL
LIN {X 0,Y 402.001,Z 477.621,A -85,B 0,C 180,E1 -11270.332,E2 -11270.332} C_VEL
LIN {X 0,Y 403.237,Z 465.295,A -85,B 0,C 180,E1 -11271.47,E2 -11271.47} C_VEL
LIN {X 0,Y 404.582,Z 451.995,A -85,B 0,C 180,E1 -11272.468,E2 -11272.468} C_VEL
LIN {X 0,Y 405.67,Z 438.143,A -85,B 0,C 180,E1 -11273.302,E2 -11273.302} C_VEL
LIN {X 0,Y 405.801,Z 434.791,A -85,B 0,C 180,E1 -11273.474,E2 -11273.474} C_VEL
LIN {X 0,Y 403.468,Z 420.647,A -85,B 0,C 180,E1 -11274.267,E2 -11274.267} C_VEL
LIN {X 0,Y 399.982,Z 405.165,A -85,B 0,C 180,E1 -11274.98,E2 -11274.98} C_VEL
LIN {X 0,Y 397.986,Z 397.296,A -85,B 0,C 180,E1 -11275.293,E2 -11275.293} C_VEL
LIN {X 0,Y 398.881,Z 388.135,A -85,B 0,C 180,E1 -11278.982,E2 -11278.982} C_VEL
LIN {X 0,Y 399.777,Z 379.601,A -85,B 0,C 180,E1 -11282.454,E2 -11282.454} C_VEL
LIN {X 0,Y 400.632,Z 372.55,A -85,B 0,C 180,E1 -11285.373,E2 -11285.373} C_VEL
LIN {X 0,Y 400.367,Z 368.451,A -85,B 0,C 180,E1 -11287.198,E2 -11287.198} C_VEL
LIN {X 0,Y 399.237,Z 362.675,A -85,B 0,C 180,E1 -11289.981,E2 -11289.981} C_VEL
LIN {X 0,Y 397.913,Z 355.632,A -85,B 0,C 180,E1 -11293.602,E2 -11293.602} C_VEL
LIN {X 0,Y 397.102,Z 351.64,A -85,B 0,C 180,E1 -11295.845,E2 -11295.845} C_VEL
LIN {X 0,Y 397.114,Z 351.635,A -85,B 0,C 180,E1 -11299.095,E2 -11299.095} C_VEL
LIN {X 0,Y 397.112,Z 351.647,A -85,B 0,C 180,E1 -11301.726,E2 -11301.726} C_VEL
LIN {X 0,Y 397.128,Z 351.646,A -85,B 0,C 180,E1 -11305.507,E2 -11305.507} C_VEL
LIN {X 0,Y 397.081,Z 351.652,A -85,B 0,C 180,E1 -11309.118,E2 -11309.118} C_VEL
LIN {X 0,Y 397.197,Z 351.634,A -85,B 0,C 180,E1 -11312.61,E2 -11312.61} C_VEL
LIN {X 0,Y 397.136,Z 351.643,A -85,B 0,C 180,E1 -11315.982,E2 -11315.982} C_VEL
LIN {X 0,Y 397.142,Z 351.641,A -85,B 0,C 180,E1 -11319.705,E2 -11319.705} C_VEL
LIN {X 0,Y 397.185,Z 351.635,A -85,B 0,C 180,E1 -11322.845,E2 -11322.845} C_VEL
LIN {X 0,Y 397.23,Z 351.626,A -85,B 0,C 180,E1 -11326.679,E2 -11326.679} C_VEL
LIN {X 0,Y 397.225,Z 351.628,A -85,B 0,C 180,E1 -11329.809,E2 -11329.809} C_VEL
LIN {X 0,Y 397.342,Z 351.616,A -85,B 0,C 180,E1 -11332.888,E2 -11332.888} C_VEL
LIN {X 0,Y 397.257,Z 351.628,A -85,B 0,C 180,E1 -11334.925,E2 -11334.925} C_VEL
LIN {X 0,Y 397.453,Z 351.599,A -85,B 0,C 180,E1 -11337.973,E2 -11337.973} C_VEL
LIN {X 0,Y 397.583,Z 351.582,A -85,B 0,C 180,E1 -11340,E2 -11340} C_VEL
LIN {X 0,Y 397.379,Z 351.613,A -85,B 0,C 180,E1 -11343.042,E2 -11343.042} C_VEL
LIN {X 0,Y 397.368,Z 351.609,A -85,B 0,C 180,E1 -11347.112,E2 -11347.112} C_VEL
LIN {X 0,Y 397.232,Z 351.629,A -85,B 0,C 180,E1 -11350.191,E2 -11350.191} C_VEL
LIN {X 0,Y 397.23,Z 351.632,A -85,B 0,C 180,E1 -11353.321,E2 -11353.321} C_VEL
LIN {X 0,Y 397.186,Z 351.633,A -85,B 0,C 180,E1 -11357.155,E2 -11357.155} C_VEL
LIN {X 0,Y 397.107,Z 351.641,A -85,B 0,C 180,E1 -11360.73,E2 -11360.73} C_VEL
LIN {X 0,Y 397.137,Z 351.636,A -85,B 0,C 180,E1 -11364.018,E2 -11364.018} C_VEL
LIN {X 0,Y 397.198,Z 351.632,A -85,B 0,C 180,E1 -11367.39,E2 -11367.39} C_VEL
LIN {X 0,Y 397.082,Z 351.647,A -85,B 0,C 180,E1 -11370.882,E2 -11370.882} C_VEL
LIN {X 0,Y 397.129,Z 351.642,A -85,B 0,C 180,E1 -11374.493,E2 -11374.493} C_VEL
LIN {X 0,Y 397.105,Z 351.645,A -85,B 0,C 180,E1 -11378.275,E2 -11378.275} C_VEL
LIN {X 0,Y 397.091,Z 351.648,A -85,B 0,C 180,E1 -11380.909,E2 -11380.909} C_VEL
LIN {X 0,Y 397.104,Z 351.648,A -85,B 0,C 180,E1 -11383.648,E2 -11383.648} C_VEL
LIN {X 0,Y 397.131,Z 351.702,A -85,B 0,C 180,E1 -11386.83,E2 -11386.83} C_VEL
LIN {X 0,Y 397.65,Z 354.975,A -85,B 0,C 180,E1 -11389.462,E2 -11389.462} C_VEL
LIN {X 0,Y 397.778,Z 358.021,A -85,B 0,C 180,E1 -11391.802,E2 -11391.802} C_VEL
LIN {X 0,Y 397.666,Z 361.518,A -85,B 0,C 180,E1 -11394.387,E2 -11394.387} C_VEL
LIN {X 0,Y 397.443,Z 364.83,A -85,B 0,C 180,E1 -11396.758,E2 -11396.758} C_VEL
LIN {X 0,Y 397.147,Z 369.898,A -85,B 0,C 180,E1 -11400.298,E2 -11400.298} C_VEL
LIN {X 0,Y 396.863,Z 375.02,A -85,B 0,C 180,E1 -11403.722,E2 -11403.722} C_VEL
LIN {X 0,Y 396.717,Z 378.49,A -85,B 0,C 180,E1 -11405.955,E2 -11405.955} C_VEL
LIN {X 0,Y 396.697,Z 380.74,A -85,B 0,C 180,E1 -11407.373,E2 -11407.373} C_VEL
LIN {X 0,Y 401.454,Z 396.164,A -85,B 0,C 180,E1 -11408.101,E2 -11408.101} C_VEL
LIN {X 0,Y 404.932,Z 409.78,A -85,B 0,C 180,E1 -11408.891,E2 -11408.891} C_VEL
LIN {X 0,Y 405.758,Z 413.736,A -85,B 0,C 180,E1 -11409.142,E2 -11409.142} C_VEL
LIN {X 0,Y 404.883,Z 427.381,A -85,B 0,C 180,E1 -11409.951,E2 -11409.951} C_VEL
LIN {X 0,Y 403.702,Z 440.495,A -85,B 0,C 180,E1 -11410.949,E2 -11410.949} C_VEL
LIN {X 0,Y 402.464,Z 452.33,A -85,B 0,C 180,E1 -11412.075,E2 -11412.075} C_VEL
LIN {X 0,Y 401.251,Z 464.067,A -85,B 0,C 180,E1 -11413.464,E2 -11413.464} C_VEL
LIN {X 0,Y 400.018,Z 474.269,A -85,B 0,C 180,E1 -11414.939,E2 -11414.939} C_VEL
LIN {X 0,Y 399.034,Z 483.134,A -85,B 0,C 180,E1 -11416.505,E2 -11416.505} C_VEL
LIN {X 0,Y 398.001,Z 491.38,A -85,B 0,C 180,E1 -11418.283,E2 -11418.283} C_VEL
LIN {X 0,Y 397.301,Z 497.14,A -85,B 0,C 180,E1 -11419.811,E2 -11419.811} C_VEL
LIN {X 0,Y 396.664,Z 503.283,A -85,B 0,C 180,E1 -11421.851,E2 -11421.851} C_VEL
LIN {X 0,Y 396.322,Z 507.851,A -85,B 0,C 180,E1 -11423.892,E2 -11423.892} C_VEL
LIN {X 0,Y 395.996,Z 511.016,A -85,B 0,C 180,E1 -11425.929,E2 -11425.929} C_VEL
LIN {X 0,Y 395.936,Z 512.878,A -85,B 0,C 180,E1 -11427.966,E2 -11427.966} C_VEL
LIN {X 0,Y 395.819,Z 513.515,A -85,B 0,C 180,E1 -11430,E2 -11430} C_VEL
LIN {X 0,Y 395.935,Z 512.939,A -85,B 0,C 180,E1 -11432.035,E2 -11432.035} C_VEL
LIN {X 0,Y 395.994,Z 511.143,A -85,B 0,C 180,E1 -11434.071,E2 -11434.071} C_VEL
LIN {X 0,Y 396.318,Z 508.041,A -85,B 0,C 180,E1 -11436.108,E2 -11436.108} C_VEL
LIN {X 0,Y 396.658,Z 503.536,A -85,B 0,C 180,E1 -11438.149,E2 -11438.149} C_VEL
LIN {X 0,Y 397.265,Z 497.472,A -85,B 0,C 180,E1 -11440.19,E2 -11440.19} C_VEL
LIN {X 0,Y 398.043,Z 490.706,A -85,B 0,C 180,E1 -11441.974,E2 -11441.974} C_VEL
LIN {X 0,Y 399.118,Z 482.303,A -85,B 0,C 180,E1 -11443.752,E2 -11443.752} C_VEL
LIN {X 0,Y 400.106,Z 473.519,A -85,B 0,C 180,E1 -11445.277,E2 -11445.277} C_VEL
LIN {X 0,Y 400.364,Z 471.155,A -85,B 0,C 180,E1 -11445.645,E2 -11445.645} C_VEL
LIN {X 0,Y 400.191,Z 467.113,A -85,B 0,C 180,E1 -11446.262,E2 -11446.262} C_VEL
LIN {X 0,Y 398.235,Z 460.444,A -85,B 0,C 180,E1 -11447.283,E2 -11447.283} C_VEL
LIN {X 0,Y 396.371,Z 453.368,A -85,B 0,C 180,E1 -11448.243,E2 -11448.243} C_VEL
LIN {X 0,Y 396.322,Z 448.676,A -85,B 0,C 180,E1 -11448.758,E2 -11448.758} C_VEL
LIN {X 0,Y 397.562,Z 436.131,A -85,B 0,C 180,E1 -11449.884,E2 -11449.884} C_VEL
LIN {X 0,Y 398.617,Z 422.685,A -85,B 0,C 180,E1 -11450.84,E2 -11450.84} C_VEL
LIN {X 0,Y 399.062,Z 414.962,A -85,B 0,C 180,E1 -11451.289,E2 -11451.289} C_VEL
LIN {X 0,Y 395.899,Z 401.29,A -85,B 0,C 180,E1 -11452.157,E2 -11452.157} C_VEL
LIN {X 0,Y 391.614,Z 386.994,A -85,B 0,C 180,E1 -11452.917,E2 -11452.917} C_VEL
LIN {X 0,Y 389.622,Z 380.899,A -85,B 0,C 180,E1 -11453.199,E2 -11453.199} C_VEL
LIN {X 0,Y 389.822,Z 377.08,A -85,B 0,C 180,E1 -11455.652,E2 -11455.652} C_VEL
LIN {X 0,Y 390.049,Z 371.958,A -85,B 0,C 180,E1 -11459.111,E2 -11459.111} C_VEL
LIN {X 0,Y 390.292,Z 367.568,A -85,B 0,C 180,E1 -11462.185,E2 -11462.185} C_VEL
LIN {X 0,Y 390.594,Z 363.464,A -85,B 0,C 180,E1 -11465.155,E2 -11465.155} C_VEL
LIN {X 0,Y 390.824,Z 360.028,A -85,B 0,C 180,E1 -11467.699,E2 -11467.699} C_VEL
LIN {X 0,Y 390.688,Z 356.577,A -85,B 0,C 180,E1 -11470.361,E2 -11470.361} C_VEL
LIN {X 0,Y 390.093,Z 352.581,A -85,B 0,C 180,E1 -11473.624,E2 -11473.624} C_VEL
LIN {X 0,Y 390.061,Z 352.521,A -85,B 0,C 180,E1 -11476.79,E2 -11476.79} C_VEL
LIN {X 0,Y 390.06,Z 352.52,A -85,B 0,C 180,E1 -11479.561,E2 -11479.561} C_VEL
LIN {X 0,Y 390.047,Z 352.522,A -85,B 0,C 180,E1 -11482.449,E2 -11482.449} C_VEL
LIN {X 0,Y 390.072,Z 352.52,A -85,B 0,C 180,E1 -11485.976,E2 -11485.976} C_VEL
LIN {X 0,Y 390.051,Z 352.524,A -85,B 0,C 180,E1 -11489.869,E2 -11489.869} C_VEL
LIN {X 0,Y 390.118,Z 352.517,A -85,B 0,C 180,E1 -11493.232,E2 -11493.232} C_VEL
LIN {X 0,Y 390.111,Z 352.516,A -85,B 0,C 180,E1 -11496.75,E2 -11496.75} C_VEL
LIN {X 0,Y 390.109,Z 352.517,A -85,B 0,C 180,E1 -11499.983,E2 -11499.983} C_VEL
LIN {X 0,Y 390.143,Z 352.514,A -85,B 0,C 180,E1 -11503.248,E2 -11503.248} C_VEL
LIN {X 0,Y 390.2,Z 352.507,A -85,B 0,C 180,E1 -11506.562,E2 -11506.562} C_VEL
LIN {X 0,Y 390.21,Z 352.501,A -85,B 0,C 180,E1 -11510.671,E2 -11510.671} C_VEL
LIN {X 0,Y 390.324,Z 352.489,A -85,B 0,C 180,E1 -11512.759,E2 -11512.759} C_VEL
LIN {X 0,Y 390.232,Z 352.498,A -85,B 0,C 180,E1 -11514.833,E2 -11514.833} C_VEL
LIN {X 0,Y 390.423,Z 352.475,A -85,B 0,C 180,E1 -11517.937,E2 -11517.937} C_VEL
LIN {X 0,Y 390.554,Z 352.463,A -85,B 0,C 180,E1 -11520,E2 -11520} C_VEL
LIN {X 0,Y 390.314,Z 352.491,A -85,B 0,C 180,E1 -11523.096,E2 -11523.096} C_VEL
LIN {X 0,Y 390.323,Z 352.49,A -85,B 0,C 180,E1 -11526.202,E2 -11526.202} C_VEL
LIN {X 0,Y 390.2,Z 352.506,A -85,B 0,C 180,E1 -11529.329,E2 -11529.329} C_VEL
LIN {X 0,Y 390.183,Z 352.51,A -85,B 0,C 180,E1 -11532.483,E2 -11532.483} C_VEL
LIN {X 0,Y 390.145,Z 352.516,A -85,B 0,C 180,E1 -11535.676,E2 -11535.676} C_VEL
LIN {X 0,Y 390.11,Z 352.52,A -85,B 0,C 180,E1 -11538.922,E2 -11538.922} C_VEL
LIN {X 0,Y 390.044,Z 352.525,A -85,B 0,C 180,E1 -11542.234,E2 -11542.234} C_VEL
LIN {X 0,Y 390.123,Z 352.516,A -85,B 0,C 180,E1 -11545.743,E2 -11545.743} C_VEL
LIN {X 0,Y 390.062,Z 352.522,A -85,B 0,C 180,E1 -11549.109,E2 -11549.109} C_VEL
LIN {X 0,Y 390.046,Z 352.528,A -85,B 0,C 180,E1 -11552.721,E2 -11552.721} C_VEL
LIN {X 0,Y 390.06,Z 352.527,A -85,B 0,C 180,E1 -11555.825,E2 -11555.825} C_VEL
LIN {X 0,Y 390.073,Z 352.521,A -85,B 0,C 180,E1 -11559.218,E2 -11559.218} C_VEL
LIN {X 0,Y 390.045,Z 352.529,A -85,B 0,C 180,E1 -11562.374,E2 -11562.374} C_VEL
LIN {X 0,Y 390.082,Z 352.615,A -85,B 0,C 180,E1 -11563.679,E2 -11563.679} C_VEL
LIN {X 0,Y 391.432,Z 359.303,A -85,B 0,C 180,E1 -11567.403,E2 -11567.403} C_VEL
LIN {X 0,Y 392.84,Z 366.804,A -85,B 0,C 180,E1 -11571.232,E2 -11571.232} C_VEL
LIN {X 0,Y 393.651,Z 371.441,A -85,B 0,C 180,E1 -11573.456,E2 -11573.456} C_VEL
LIN {X 0,Y 393.506,Z 375.504,A -85,B 0,C 180,E1 -11575.241,E2 -11575.241} C_VEL
LIN {X 0,Y 392.46,Z 383.742,A -85,B 0,C 180,E1 -11578.713,E2 -11578.713} C_VEL
LIN {X 0,Y 391.506,Z 392.142,A -85,B 0,C 180,E1 -11582.177,E2 -11582.177} C_VEL
LIN {X 0,Y 391.032,Z 397.251,A -85,B 0,C 180,E1 -11584.257,E2 -11584.257} C_VEL
LIN {X 0,Y 395.025,Z 413.204,A -85,B 0,C 180,E1 -11584.937,E2 -11584.937} C_VEL
LIN {X 0,Y 397.915,Z 427.798,A -85,B 0,C 180,E1 -11585.709,E2 -11585.709} C_VEL
LIN {X 0,Y 399.145,Z 437.561,A -85,B 0,C 180,E1 -11586.29,E2 -11586.29} C_VEL
LIN {X 0,Y 398,Z 451.541,A -85,B 0,C 180,E1 -11587.14,E2 -11587.14} C_VEL
LIN {X 0,Y 396.65,Z 464.872,A -85,B 0,C 180,E1 -11588.155,E2 -11588.155} C_VEL
LIN {X 0,Y 395.235,Z 477.204,A -85,B 0,C 180,E1 -11589.303,E2 -11589.303} C_VEL
LIN {X 0,Y 393.853,Z 489.806,A -85,B 0,C 180,E1 -11590.724,E2 -11590.724} C_VEL
LIN {X 0,Y 392.596,Z 501.28,A -85,B 0,C 180,E1 -11592.282,E2 -11592.282} C_VEL
LIN {X 0,Y 391.456,Z 510.945,A -85,B 0,C 180,E1 -11593.842,E2 -11593.842} C_VEL
LIN {X 0,Y 390.507,Z 520.467,A -85,B 0,C 180,E1 -11595.672,E2 -11595.672} C_VEL
LIN {X 0,Y 389.78,Z 528.394,A -85,B 0,C 180,E1 -11597.504,E2 -11597.504} C_VEL
LIN {X 0,Y 389.343,Z 534.13,A -85,B 0,C 180,E1 -11599.074,E2 -11599.074} C_VEL
LIN {X 0,Y 388.951,Z 540.351,A -85,B 0,C 180,E1 -11601.165,E2 -11601.165} C_VEL
LIN {X 0,Y 388.779,Z 545.14,A -85,B 0,C 180,E1 -11603.252,E2 -11603.252} C_VEL
LIN {X 0,Y 388.717,Z 547.806,A -85,B 0,C 180,E1 -11604.813,E2 -11604.813} C_VEL
LIN {X 0,Y 388.676,Z 550.295,A -85,B 0,C 180,E1 -11606.89,E2 -11606.89} C_VEL
LIN {X 0,Y 388.779,Z 551.08,A -85,B 0,C 180,E1 -11607.928,E2 -11607.928} C_VEL
LIN {X 0,Y 388.743,Z 551.714,A -85,B 0,C 180,E1 -11610,E2 -11610} C_VEL
LIN {X 0,Y 388.779,Z 551.075,A -85,B 0,C 180,E1 -11612.072,E2 -11612.072} C_VEL
LIN {X 0,Y 388.699,Z 549.197,A -85,B 0,C 180,E1 -11614.147,E2 -11614.147} C_VEL
LIN {X 0,Y 388.796,Z 546.076,A -85,B 0,C 180,E1 -11616.226,E2 -11616.226} C_VEL
LIN {X 0,Y 388.91,Z 541.637,A -85,B 0,C 180,E1 -11618.312,E2 -11618.312} C_VEL
LIN {X 0,Y 389.165,Z 535.779,A -85,B 0,C 180,E1 -11620.404,E2 -11620.404} C_VEL
LIN {X 0,Y 389.679,Z 529.402,A -85,B 0,C 180,E1 -11622.235,E2 -11622.235} C_VEL
LIN {X 0,Y 390.404,Z 521.696,A -85,B 0,C 180,E1 -11624.065,E2 -11624.065} C_VEL
LIN {X 0,Y 391.297,Z 512.42,A -85,B 0,C 180,E1 -11625.897,E2 -11625.897} C_VEL
LIN {X 0,Y 392.553,Z 501.232,A -85,B 0,C 180,E1 -11627.719,E2 -11627.719} C_VEL
LIN {X 0,Y 393.837,Z 489.756,A -85,B 0,C 180,E1 -11629.276,E2 -11629.276} C_VEL
LIN {X 0,Y 395.249,Z 477.146,A -85,B 0,C 180,E1 -11630.696,E2 -11630.696} C_VEL
LIN {X 0,Y 396.569,Z 464.778,A -85,B 0,C 180,E1 -11631.849,E2 -11631.849} C_VEL
LIN {X 0,Y 397.989,Z 451.427,A -85,B 0,C 180,E1 -11632.861,E2 -11632.861} C_VEL
LIN {X 0,Y 399.161,Z 436.604,A -85,B 0,C 180,E1 -11633.754,E2 -11633.754} C_VEL
LIN {X 0,Y 397.287,Z 424.29,A -85,B 0,C 180,E1 -11634.484,E2 -11634.484} C_VEL
LIN {X 0,Y 394.312,Z 410.181,A -85,B 0,C 180,E1 -11635.195,E2 -11635.195} C_VEL
LIN {X 0,Y 391.049,Z 397.106,A -85,B 0,C 180,E1 -11635.76,E2 -11635.76} C_VEL
LIN {X 0,Y 391.846,Z 389.326,A -85,B 0,C 180,E1 -11638.964,E2 -11638.964} C_VEL
LIN {X 0,Y 392.775,Z 380.91,A -85,B 0,C 180,E1 -11642.466,E2 -11642.466} C_VEL
LIN {X 0,Y 393.687,Z 373.798,A -85,B 0,C 180,E1 -11645.463,E2 -11645.463} C_VEL
LIN {X 0,Y 393.359,Z 369.55,A -85,B 0,C 180,E1 -11647.407,E2 -11647.407} C_VEL
LIN {X 0,Y 392.283,Z 363.945,A -85,B 0,C 180,E1 -11650.163,E2 -11650.163} C_VEL
LIN {X 0,Y 391.256,Z 358.424,A -85,B 0,C 180,E1 -11653.046,E2 -11653.046} C_VEL
LIN {X 0,Y 390.07,Z 352.517,A -85,B 0,C 180,E1 -11656.444,E2 -11656.444} C_VEL
LIN {X 0,Y 390.077,Z 352.515,A -85,B 0,C 180,E1 -11659.563,E2 -11659.563} C_VEL
LIN {X 0,Y 390.049,Z 352.527,A -85,B 0,C 180,E1 -11662.449,E2 -11662.449} C_VEL
LIN {X 0,Y 390.086,Z 352.524,A -85,B 0,C 180,E1 -11666.047,E2 -11666.047} C_VEL
LIN {X 0,Y 390.049,Z 352.526,A -85,B 0,C 180,E1 -11669.869,E2 -11669.869} C_VEL
LIN {X 0,Y 390.116,Z 352.519,A -85,B 0,C 180,E1 -11673.232,E2 -11673.232} C_VEL
LIN {X 0,Y 390.109,Z 352.516,A -85,B 0,C 180,E1 -11676.75,E2 -11676.75} C_VEL
LIN {X 0,Y 390.107,Z 352.518,A -85,B 0,C 180,E1 -11679.983,E2 -11679.983} C_VEL
LIN {X 0,Y 390.141,Z 352.511,A -85,B 0,C 180,E1 -11683.249,E2 -11683.249} C_VEL
LIN {X 0,Y 390.198,Z 352.503,A -85,B 0,C 180,E1 -11686.562,E2 -11686.562} C_VEL
LIN {X 0,Y 390.176,Z 352.507,A -85,B 0,C 180,E1 -11689.623,E2 -11689.623} C_VEL
LIN {X 0,Y 390.289,Z 352.494,A -85,B 0,C 180,E1 -11692.759,E2 -11692.759} C_VEL
LIN {X 0,Y 390.228,Z 352.502,A -85,B 0,C 180,E1 -11694.834,E2 -11694.834} C_VEL
LIN {X 0,Y 390.422,Z 352.475,A -85,B 0,C 180,E1 -11697.937,E2 -11697.937} C_VEL
LIN {X 0,Y 390.553,Z 352.458,A -85,B 0,C 180,E1 -11700,E2 -11700} C_VEL
LIN {X 0,Y 390.314,Z 352.492,A -85,B 0,C 180,E1 -11703.097,E2 -11703.097} C_VEL
LIN {X 0,Y 390.314,Z 352.487,A -85,B 0,C 180,E1 -11706.654,E2 -11706.654} C_VEL
LIN {X 0,Y 390.214,Z 352.502,A -85,B 0,C 180,E1 -11709.329,E2 -11709.329} C_VEL
LIN {X 0,Y 390.182,Z 352.506,A -85,B 0,C 180,E1 -11712.483,E2 -11712.483} C_VEL
LIN {X 0,Y 390.144,Z 352.511,A -85,B 0,C 180,E1 -11715.677,E2 -11715.677} C_VEL
LIN {X 0,Y 390.11,Z 352.516,A -85,B 0,C 180,E1 -11718.922,E2 -11718.922} C_VEL
LIN {X 0,Y 390.044,Z 352.525,A -85,B 0,C 180,E1 -11722.234,E2 -11722.234} C_VEL
LIN {X 0,Y 390.123,Z 352.514,A -85,B 0,C 180,E1 -11725.744,E2 -11725.744} C_VEL
LIN {X 0,Y 390.062,Z 352.519,A -85,B 0,C 180,E1 -11729.109,E2 -11729.109} C_VEL
LIN {X 0,Y 390.046,Z 352.523,A -85,B 0,C 180,E1 -11732.721,E2 -11732.721} C_VEL
LIN {X 0,Y 390.059,Z 352.523,A -85,B 0,C 180,E1 -11735.825,E2 -11735.825} C_VEL
LIN {X 0,Y 390.072,Z 352.522,A -85,B 0,C 180,E1 -11739.218,E2 -11739.218} C_VEL
LIN {X 0,Y 390.046,Z 352.526,A -85,B 0,C 180,E1 -11742.374,E2 -11742.374} C_VEL
LIN {X 0,Y 390.047,Z 352.528,A -85,B 0,C 180,E1 -11745.354,E2 -11745.354} C_VEL
LIN {X 0,Y 390.069,Z 352.542,A -85,B 0,C 180,E1 -11746.454,E2 -11746.454} C_VEL
LIN {X 0,Y 390.672,Z 356.432,A -85,B 0,C 180,E1 -11749.637,E2 -11749.637} C_VEL
LIN {X 0,Y 390.78,Z 359.883,A -85,B 0,C 180,E1 -11752.309,E2 -11752.309} C_VEL
LIN {X 0,Y 390.604,Z 363.296,A -85,B 0,C 180,E1 -11754.847,E2 -11754.847} C_VEL
LIN {X 0,Y 390.257,Z 368.371,A -85,B 0,C 180,E1 -11758.516,E2 -11758.516} C_VEL
LIN {X 0,Y 389.964,Z 373.499,A -85,B 0,C 180,E1 -11762.058,E2 -11762.058} C_VEL
LIN {X 0,Y 389.735,Z 378.71,A -85,B 0,C 180,E1 -11765.496,E2 -11765.496} C_VEL
LIN {X 0,Y 389.657,Z 380.905,A -85,B 0,C 180,E1 -11766.905,E2 -11766.905} C_VEL
LIN {X 0,Y 394.789,Z 397.314,A -85,B 0,C 180,E1 -11767.719,E2 -11767.719} C_VEL
LIN {X 0,Y 398.302,Z 411.168,A -85,B 0,C 180,E1 -11768.557,E2 -11768.557} C_VEL
LIN {X 0,Y 399.149,Z 415.763,A -85,B 0,C 180,E1 -11768.861,E2 -11768.861} C_VEL
LIN {X 0,Y 398.26,Z 427.93,A -85,B 0,C 180,E1 -11769.603,E2 -11769.603} C_VEL
LIN {X 0,Y 397.009,Z 440.987,A -85,B 0,C 180,E1 -11770.615,E2 -11770.615} C_VEL
LIN {X 0,Y 395.733,Z 452.78,A -85,B 0,C 180,E1 -11771.759,E2 -11771.759} C_VEL
LIN {X 0,Y 394.459,Z 464.489,A -85,B 0,C 180,E1 -11773.171,E2 -11773.171} C_VEL
LIN {X 0,Y 393.131,Z 474.938,A -85,B 0,C 180,E1 -11774.713,E2 -11774.713} C_VEL
LIN {X 0,Y 392.127,Z 483.52,A -85,B 0,C 180,E1 -11776.262,E2 -11776.262} C_VEL
LIN {X 0,Y 391.019,Z 491.755,A -85,B 0,C 180,E1 -11778.071,E2 -11778.071} C_VEL
LIN {X 0,Y 390.317,Z 497.504,A -85,B 0,C 180,E1 -11779.627,E2 -11779.627} C_VEL
LIN {X 0,Y 389.648,Z 503.64,A -85,B 0,C 180,E1 -11781.704,E2 -11781.704} C_VEL
LIN {X 0,Y 389.26,Z 508.203,A -85,B 0,C 180,E1 -11783.781,E2 -11783.781} C_VEL
LIN {X 0,Y 388.915,Z 511.365,A -85,B 0,C 180,E1 -11785.855,E2 -11785.855} C_VEL
LIN {X 0,Y 388.871,Z 513.223,A -85,B 0,C 180,E1 -11787.929,E2 -11787.929} C_VEL
LIN {X 0,Y 388.746,Z 513.86,A -85,B 0,C 180,E1 -11790,E2 -11790} C_VEL
LIN {X 0,Y 388.871,Z 513.283,A -85,B 0,C 180,E1 -11792.072,E2 -11792.072} C_VEL
LIN {X 0,Y 388.913,Z 511.49,A -85,B 0,C 180,E1 -11794.145,E2 -11794.145} C_VEL
LIN {X 0,Y 389.256,Z 508.391,A -85,B 0,C 180,E1 -11796.219,E2 -11796.219} C_VEL
LIN {X 0,Y 389.641,Z 503.891,A -85,B 0,C 180,E1 -11798.297,E2 -11798.297} C_VEL
LIN {X 0,Y 390.279,Z 497.833,A -85,B 0,C 180,E1 -11800.374,E2 -11800.374} C_VEL
LIN {X 0,Y 391.076,Z 491.076,A -85,B 0,C 180,E1 -11802.19,E2 -11802.19} C_VEL
LIN {X 0,Y 392.232,Z 482.683,A -85,B 0,C 180,E1 -11803.999,E2 -11803.999} C_VEL
LIN {X 0,Y 393.267,Z 473.914,A -85,B 0,C 180,E1 -11805.549,E2 -11805.549} C_VEL
LIN {X 0,Y 394.38,Z 465.197,A -85,B 0,C 180,E1 -11806.833,E2 -11806.833} C_VEL
LIN {X 0,Y 395.552,Z 454.798,A -85,B 0,C 180,E1 -11808.116,E2 -11808.116} C_VEL
LIN {X 0,Y 396.322,Z 448.676,A -85,B 0,C 180,E1 -11808.758,E2 -11808.758} C_VEL
LIN {X 0,Y 396.267,Z 443.896,A -85,B 0,C 180,E1 -11809.251,E2 -11809.251} C_VEL
LIN {X 0,Y 394.347,Z 436,A -85,B 0,C 180,E1 -11810.085,E2 -11810.085} C_VEL
LIN {X 0,Y 392.356,Z 427.877,A -85,B 0,C 180,E1 -11810.86,E2 -11810.86} C_VEL
LIN {X 0,Y 392.097,Z 422.618,A -85,B 0,C 180,E1 -11811.246,E2 -11811.246} C_VEL
LIN {X 0,Y 392.475,Z 417.41,A -85,B 0,C 180,E1 -11811.555,E2 -11811.555} C_VEL
LIN {X 0,Y 390.636,Z 407.912,A -85,B 0,C 180,E1 -11812.199,E2 -11812.199} C_VEL
LIN {X 0,Y 386.671,Z 393.488,A -85,B 0,C 180,E1 -11813.057,E2 -11813.057} C_VEL
LIN {X 0,Y 382.621,Z 381.062,A -85,B 0,C 180,E1 -11813.685,E2 -11813.685} C_VEL
LIN {X 0,Y 382.793,Z 377.306,A -85,B 0,C 180,E1 -11816.145,E2 -11816.145} C_VEL
LIN {X 0,Y 383.067,Z 372.147,A -85,B 0,C 180,E1 -11819.694,E2 -11819.694} C_VEL
LIN {X 0,Y 383.386,Z 367.027,A -85,B 0,C 180,E1 -11823.363,E2 -11823.363} C_VEL
LIN {X 0,Y 383.698,Z 363.065,A -85,B 0,C 180,E1 -11826.3,E2 -11826.3} C_VEL
LIN {X 0,Y 383.827,Z 360.179,A -85,B 0,C 180,E1 -11828.503,E2 -11828.503} C_VEL
LIN {X 0,Y 383.549,Z 356.667,A -85,B 0,C 180,E1 -11831.299,E2 -11831.299} C_VEL
LIN {X 0,Y 383.004,Z 353.403,A -85,B 0,C 180,E1 -11834.127,E2 -11834.127} C_VEL
LIN {X 0,Y 383.014,Z 353.397,A -85,B 0,C 180,E1 -11837.24,E2 -11837.24} C_VEL
LIN {X 0,Y 383.019,Z 353.396,A -85,B 0,C 180,E1 -11840.414,E2 -11840.414} C_VEL
LIN {X 0,Y 383.029,Z 353.398,A -85,B 0,C 180,E1 -11844.045,E2 -11844.045} C_VEL
LIN {X 0,Y 382.991,Z 353.402,A -85,B 0,C 180,E1 -11847.578,E2 -11847.578} C_VEL
LIN {X 0,Y 382.997,Z 353.404,A -85,B 0,C 180,E1 -11850.3,E2 -11850.3} C_VEL
LIN {X 0,Y 383.061,Z 353.394,A -85,B 0,C 180,E1 -11852.698,E2 -11852.698} C_VEL
LIN {X 0,Y 383.057,Z 353.398,A -85,B 0,C 180,E1 -11855.04,E2 -11855.04} C_VEL
LIN {X 0,Y 382.998,Z 353.401,A -85,B 0,C 180,E1 -11858.469,E2 -11858.469} C_VEL
LIN {X 0,Y 383.068,Z 353.391,A -85,B 0,C 180,E1 -11861.826,E2 -11861.826} C_VEL
LIN {X 0,Y 383.115,Z 353.385,A -85,B 0,C 180,E1 -11865.118,E2 -11865.118} C_VEL
LIN {X 0,Y 383.103,Z 353.387,A -85,B 0,C 180,E1 -11868.358,E2 -11868.358} C_VEL
LIN {X 0,Y 383.309,Z 353.362,A -85,B 0,C 180,E1 -11871.933,E2 -11871.933} C_VEL
LIN {X 0,Y 383.204,Z 353.373,A -85,B 0,C 180,E1 -11874.738,E2 -11874.738} C_VEL
LIN {X 0,Y 383.391,Z 353.351,A -85,B 0,C 180,E1 -11877.899,E2 -11877.899} C_VEL
LIN {X 0,Y 383.523,Z 353.339,A -85,B 0,C 180,E1 -11880,E2 -11880} C_VEL
LIN {X 0,Y 383.251,Z 353.371,A -85,B 0,C 180,E1 -11883.153,E2 -11883.153} C_VEL
LIN {X 0,Y 383.277,Z 353.368,A -85,B 0,C 180,E1 -11886.316,E2 -11886.316} C_VEL
LIN {X 0,Y 383.15,Z 353.384,A -85,B 0,C 180,E1 -11889.502,E2 -11889.502} C_VEL
LIN {X 0,Y 383.146,Z 353.386,A -85,B 0,C 180,E1 -11892.716,E2 -11892.716} C_VEL
LIN {X 0,Y 383.086,Z 353.394,A -85,B 0,C 180,E1 -11895.973,E2 -11895.973} C_VEL
LIN {X 0,Y 383.065,Z 353.395,A -85,B 0,C 180,E1 -11899.283,E2 -11899.283} C_VEL
LIN {X 0,Y 383.042,Z 353.398,A -85,B 0,C 180,E1 -11903.451,E2 -11903.451} C_VEL
LIN {X 0,Y 383.083,Z 353.392,A -85,B 0,C 180,E1 -11906.123,E2 -11906.123} C_VEL
LIN {X 0,Y 383.044,Z 353.398,A -85,B 0,C 180,E1 -11908.492,E2 -11908.492} C_VEL
LIN {X 0,Y 383.012,Z 353.401,A -85,B 0,C 180,E1 -11912.149,E2 -11912.149} C_VEL
LIN {X 0,Y 383.021,Z 353.402,A -85,B 0,C 180,E1 -11914.667,E2 -11914.667} C_VEL
LIN {X 0,Y 383.004,Z 353.404,A -85,B 0,C 180,E1 -11917.904,E2 -11917.904} C_VEL
LIN {X 0,Y 382.986,Z 353.405,A -85,B 0,C 180,E1 -11921.347,E2 -11921.347} C_VEL
LIN {X 0,Y 383.038,Z 353.542,A -85,B 0,C 180,E1 -11923.114,E2 -11923.114} C_VEL
LIN {X 0,Y 384.413,Z 360.285,A -85,B 0,C 180,E1 -11926.995,E2 -11926.995} C_VEL
LIN {X 0,Y 385.841,Z 367.974,A -85,B 0,C 180,E1 -11931.008,E2 -11931.008} C_VEL
LIN {X 0,Y 386.612,Z 372.3,A -85,B 0,C 180,E1 -11933.138,E2 -11933.138} C_VEL
LIN {X 0,Y 386.619,Z 376.109,A -85,B 0,C 180,E1 -11934.886,E2 -11934.886} C_VEL
LIN {X 0,Y 385.643,Z 383.558,A -85,B 0,C 180,E1 -11938.096,E2 -11938.096} C_VEL
LIN {X 0,Y 384.621,Z 391.919,A -85,B 0,C 180,E1 -11941.635,E2 -11941.635} C_VEL
LIN {X 0,Y 384.091,Z 396.965,A -85,B 0,C 180,E1 -11943.771,E2 -11943.771} C_VEL
LIN {X 0,Y 388.433,Z 414.281,A -85,B 0,C 180,E1 -11944.55,E2 -11944.55} C_VEL
LIN {X 0,Y 391.319,Z 429.044,A -85,B 0,C 180,E1 -11945.367,E2 -11945.367} C_VEL
LIN {X 0,Y 392.456,Z 438.597,A -85,B 0,C 180,E1 -11945.964,E2 -11945.964} C_VEL
LIN {X 0,Y 391.228,Z 452.785,A -85,B 0,C 180,E1 -11946.861,E2 -11946.861} C_VEL
LIN {X 0,Y 389.855,Z 465.87,A -85,B 0,C 180,E1 -11947.894,E2 -11947.894} C_VEL
LIN {X 0,Y 388.294,Z 479.231,A -85,B 0,C 180,E1 -11949.194,E2 -11949.194} C_VEL
LIN {X 0,Y 386.834,Z 491.434,A -85,B 0,C 180,E1 -11950.636,E2 -11950.636} C_VEL
LIN {X 0,Y 385.541,Z 502.605,A -85,B 0,C 180,E1 -11952.221,E2 -11952.221} C_VEL
LIN {X 0,Y 384.392,Z 512.061,A -85,B 0,C 180,E1 -11953.81,E2 -11953.81} C_VEL
LIN {X 0,Y 383.432,Z 521.347,A -85,B 0,C 180,E1 -11955.673,E2 -11955.673} C_VEL
LIN {X 0,Y 382.673,Z 529.06,A -85,B 0,C 180,E1 -11957.538,E2 -11957.538} C_VEL
LIN {X 0,Y 382.124,Z 535.434,A -85,B 0,C 180,E1 -11959.402,E2 -11959.402} C_VEL
LIN {X 0,Y 381.82,Z 541.289,A -85,B 0,C 180,E1 -11961.532,E2 -11961.532} C_VEL
LIN {X 0,Y 381.697,Z 545.734,A -85,B 0,C 180,E1 -11963.657,E2 -11963.657} C_VEL
LIN {X 0,Y 381.621,Z 548.861,A -85,B 0,C 180,E1 -11965.775,E2 -11965.775} C_VEL
LIN {X 0,Y 381.678,Z 550.734,A -85,B 0,C 180,E1 -11967.889,E2 -11967.889} C_VEL
LIN {X 0,Y 381.672,Z 551.37,A -85,B 0,C 180,E1 -11970,E2 -11970} C_VEL
LIN {X 0,Y 381.679,Z 550.729,A -85,B 0,C 180,E1 -11972.11,E2 -11972.11} C_VEL
LIN {X 0,Y 381.623,Z 548.85,A -85,B 0,C 180,E1 -11974.224,E2 -11974.224} C_VEL
LIN {X 0,Y 381.706,Z 545.723,A -85,B 0,C 180,E1 -11976.342,E2 -11976.342} C_VEL
LIN {X 0,Y 381.82,Z 541.278,A -85,B 0,C 180,E1 -11978.468,E2 -11978.468} C_VEL
LIN {X 0,Y 382.124,Z 535.414,A -85,B 0,C 180,E1 -11980.598,E2 -11980.598} C_VEL
LIN {X 0,Y 382.666,Z 529.028,A -85,B 0,C 180,E1 -11982.462,E2 -11982.462} C_VEL
LIN {X 0,Y 383.431,Z 521.311,A -85,B 0,C 180,E1 -11984.326,E2 -11984.326} C_VEL
LIN {X 0,Y 384.39,Z 512.023,A -85,B 0,C 180,E1 -11986.19,E2 -11986.19} C_VEL
LIN {X 0,Y 385.501,Z 502.557,A -85,B 0,C 180,E1 -11987.78,E2 -11987.78} C_VEL
LIN {X 0,Y 386.952,Z 490.384,A -85,B 0,C 180,E1 -11989.496,E2 -11989.496} C_VEL
LIN {X 0,Y 388.408,Z 477.967,A -85,B 0,C 180,E1 -11990.938,E2 -11990.938} C_VEL
LIN {X 0,Y 389.941,Z 464.265,A -85,B 0,C 180,E1 -11992.24,E2 -11992.24} C_VEL
LIN {X 0,Y 391.412,Z 450.85,A -85,B 0,C 180,E1 -11993.267,E2 -11993.267} C_VEL
LIN {X 0,Y 392.516,Z 437.856,A -85,B 0,C 180,E1 -11994.07,E2 -11994.07} C_VEL
LIN {X 0,Y 390.47,Z 424.265,A -85,B 0,C 180,E1 -11994.903,E2 -11994.903} C_VEL
LIN {X 0,Y 387.21,Z 409.051,A -85,B 0,C 180,E1 -11995.691,E2 -11995.691} C_VEL
LIN {X 0,Y 384.092,Z 396.968,A -85,B 0,C 180,E1 -11996.214,E2 -11996.214} C_VEL
LIN {X 0,Y 384.937,Z 389.112,A -85,B 0,C 180,E1 -11999.535,E2 -11999.535} C_VEL
LIN {X 0,Y 385.998,Z 380.728,A -85,B 0,C 180,E1 -12003.108,E2 -12003.108} C_VEL
LIN {X 0,Y 386.734,Z 375.072,A -85,B 0,C 180,E1 -12005.558,E2 -12005.558} C_VEL
LIN {X 0,Y 386.397,Z 370.84,A -85,B 0,C 180,E1 -12007.54,E2 -12007.54} C_VEL
LIN {X 0,Y 385.016,Z 363.824,A -85,B 0,C 180,E1 -12011.082,E2 -12011.082} C_VEL
LIN {X 0,Y 383.996,Z 358.336,A -85,B 0,C 180,E1 -12014.066,E2 -12014.066} C_VEL
LIN {X 0,Y 383.033,Z 353.398,A -85,B 0,C 180,E1 -12016.984,E2 -12016.984} C_VEL
LIN {X 0,Y 383.024,Z 353.401,A -85,B 0,C 180,E1 -12020.412,E2 -12020.412} C_VEL
LIN {X 0,Y 383.029,Z 353.403,A -85,B 0,C 180,E1 -12024.045,E2 -12024.045} C_VEL
LIN {X 0,Y 382.989,Z 353.41,A -85,B 0,C 180,E1 -12027.578,E2 -12027.578} C_VEL
LIN {X 0,Y 382.994,Z 353.404,A -85,B 0,C 180,E1 -12030.3,E2 -12030.3} C_VEL
LIN {X 0,Y 383.059,Z 353.395,A -85,B 0,C 180,E1 -12032.698,E2 -12032.698} C_VEL
LIN {X 0,Y 383.036,Z 353.398,A -85,B 0,C 180,E1 -12036.193,E2 -12036.193} C_VEL
LIN {X 0,Y 383.058,Z 353.394,A -85,B 0,C 180,E1 -12039.599,E2 -12039.599} C_VEL
LIN {X 0,Y 383.108,Z 353.39,A -85,B 0,C 180,E1 -12042.932,E2 -12042.932} C_VEL
LIN {X 0,Y 383.129,Z 353.384,A -85,B 0,C 180,E1 -12046.464,E2 -12046.464} C_VEL
LIN {X 0,Y 383.14,Z 353.385,A -85,B 0,C 180,E1 -12049.43,E2 -12049.43} C_VEL
LIN {X 0,Y 383.237,Z 353.372,A -85,B 0,C 180,E1 -12052.625,E2 -12052.625} C_VEL
LIN {X 0,Y 383.2,Z 353.377,A -85,B 0,C 180,E1 -12054.739,E2 -12054.739} C_VEL
LIN {X 0,Y 383.389,Z 353.35,A -85,B 0,C 180,E1 -12057.899,E2 -12057.899} C_VEL
LIN {X 0,Y 383.522,Z 353.333,A -85,B 0,C 180,E1 -12060,E2 -12060} C_VEL
LIN {X 0,Y 383.25,Z 353.371,A -85,B 0,C 180,E1 -12063.154,E2 -12063.154} C_VEL
LIN {X 0,Y 383.273,Z 353.366,A -85,B 0,C 180,E1 -12066.649,E2 -12066.649} C_VEL
LIN {X 0,Y 383.265,Z 353.367,A -85,B 0,C 180,E1 -12068.436,E2 -12068.436} C_VEL
LIN {X 0,Y 383.111,Z 353.385,A -85,B 0,C 180,E1 -12071.642,E2 -12071.642} C_VEL
LIN {X 0,Y 383.116,Z 353.384,A -85,B 0,C 180,E1 -12074.882,E2 -12074.882} C_VEL
LIN {X 0,Y 383.093,Z 353.387,A -85,B 0,C 180,E1 -12078.172,E2 -12078.172} C_VEL
LIN {X 0,Y 382.997,Z 353.399,A -85,B 0,C 180,E1 -12081.531,E2 -12081.531} C_VEL
LIN {X 0,Y 383.056,Z 353.393,A -85,B 0,C 180,E1 -12084.96,E2 -12084.96} C_VEL
LIN {X 0,Y 383.044,Z 353.398,A -85,B 0,C 180,E1 -12088.493,E2 -12088.493} C_VEL
LIN {X 0,Y 383.013,Z 353.401,A -85,B 0,C 180,E1 -12092.15,E2 -12092.15} C_VEL
LIN {X 0,Y 383.021,Z 353.4,A -85,B 0,C 180,E1 -12094.668,E2 -12094.668} C_VEL
LIN {X 0,Y 383.002,Z 353.402,A -85,B 0,C 180,E1 -12097.904,E2 -12097.904} C_VEL
LIN {X 0,Y 382.987,Z 353.405,A -85,B 0,C 180,E1 -12101.347,E2 -12101.347} C_VEL
LIN {X 0,Y 382.999,Z 353.404,A -85,B 0,C 180,E1 -12104.303,E2 -12104.303} C_VEL
LIN {X 0,Y 383.051,Z 353.614,A -85,B 0,C 180,E1 -12106.26,E2 -12106.26} C_VEL
LIN {X 0,Y 383.545,Z 356.539,A -85,B 0,C 180,E1 -12108.726,E2 -12108.726} C_VEL
LIN {X 0,Y 383.773,Z 360,A -85,B 0,C 180,E1 -12111.491,E2 -12111.491} C_VEL
LIN {X 0,Y 383.651,Z 363.439,A -85,B 0,C 180,E1 -12114.112,E2 -12114.112} C_VEL
LIN {X 0,Y 383.32,Z 368.027,A -85,B 0,C 180,E1 -12117.5,E2 -12117.5} C_VEL
LIN {X 0,Y 383.055,Z 371.972,A -85,B 0,C 180,E1 -12120.305,E2 -12120.305} C_VEL
LIN {X 0,Y 382.807,Z 377.533,A -85,B 0,C 180,E1 -12124.106,E2 -12124.106} C_VEL
LIN {X 0,Y 382.637,Z 381.095,A -85,B 0,C 180,E1 -12126.436,E2 -12126.436} C_VEL
LIN {X 0,Y 385.241,Z 389.07,A -85,B 0,C 180,E1 -12126.813,E2 -12126.813} C_VEL
LIN {X 0,Y 389.441,Z 403.22,A -85,B 0,C 180,E1 -12127.608,E2 -12127.608} C_VEL
LIN {X 0,Y 392.518,Z 416.522,A -85,B 0,C 180,E1 -12128.494,E2 -12128.494} C_VEL
LIN {X 0,Y 391.657,Z 428.476,A -85,B 0,C 180,E1 -12129.243,E2 -12129.243} C_VEL
LIN {X 0,Y 390.349,Z 441.476,A -85,B 0,C 180,E1 -12130.27,E2 -12130.27} C_VEL
LIN {X 0,Y 389.022,Z 453.229,A -85,B 0,C 180,E1 -12131.433,E2 -12131.433} C_VEL
LIN {X 0,Y 387.68,Z 464.909,A -85,B 0,C 180,E1 -12132.867,E2 -12132.867} C_VEL
LIN {X 0,Y 386.256,Z 475.568,A -85,B 0,C 180,E1 -12134.473,E2 -12134.473} C_VEL
LIN {X 0,Y 385.224,Z 483.904,A -85,B 0,C 180,E1 -12136.011,E2 -12136.011} C_VEL
LIN {X 0,Y 384.07,Z 492.128,A -85,B 0,C 180,E1 -12137.852,E2 -12137.852} C_VEL
LIN {X 0,Y 383.34,Z 497.867,A -85,B 0,C 180,E1 -12139.436,E2 -12139.436} C_VEL
LIN {X 0,Y 382.607,Z 503.998,A -85,B 0,C 180,E1 -12141.55,E2 -12141.55} C_VEL
LIN {X 0,Y 382.204,Z 508.555,A -85,B 0,C 180,E1 -12143.666,E2 -12143.666} C_VEL
LIN {X 0,Y 381.838,Z 511.714,A -85,B 0,C 180,E1 -12145.778,E2 -12145.778} C_VEL
LIN {X 0,Y 381.808,Z 513.568,A -85,B 0,C 180,E1 -12147.89,E2 -12147.89} C_VEL
LIN {X 0,Y 381.676,Z 514.204,A -85,B 0,C 180,E1 -12150,E2 -12150} C_VEL
LIN {X 0,Y 381.808,Z 513.627,A -85,B 0,C 180,E1 -12152.11,E2 -12152.11} C_VEL
LIN {X 0,Y 381.836,Z 511.836,A -85,B 0,C 180,E1 -12154.222,E2 -12154.222} C_VEL
LIN {X 0,Y 382.201,Z 508.741,A -85,B 0,C 180,E1 -12156.334,E2 -12156.334} C_VEL
LIN {X 0,Y 382.597,Z 504.246,A -85,B 0,C 180,E1 -12158.451,E2 -12158.451} C_VEL
LIN {X 0,Y 383.304,Z 498.193,A -85,B 0,C 180,E1 -12160.565,E2 -12160.565} C_VEL
LIN {X 0,Y 384.136,Z 491.444,A -85,B 0,C 180,E1 -12162.414,E2 -12162.414} C_VEL
LIN {X 0,Y 385.357,Z 483.061,A -85,B 0,C 180,E1 -12164.253,E2 -12164.253} C_VEL
LIN {X 0,Y 386.411,Z 474.309,A -85,B 0,C 180,E1 -12165.832,E2 -12165.832} C_VEL
LIN {X 0,Y 387.853,Z 463.672,A -85,B 0,C 180,E1 -12167.397,E2 -12167.397} C_VEL
LIN {X 0,Y 389.134,Z 452.893,A -85,B 0,C 180,E1 -12168.698,E2 -12168.698} C_VEL
LIN {X 0,Y 390.437,Z 441.076,A -85,B 0,C 180,E1 -12169.862,E2 -12169.862} C_VEL
LIN {X 0,Y 391.569,Z 429.064,A -85,B 0,C 180,E1 -12170.817,E2 -12170.817} C_VEL
LIN {X 0,Y 392.097,Z 422.618,A -85,B 0,C 180,E1 -12171.246,E2 -12171.246} C_VEL
LIN {X 0,Y 391.905,Z 419.104,A -85,B 0,C 180,E1 -12171.492,E2 -12171.492} C_VEL
LIN {X 0,Y 390.937,Z 415.779,A -85,B 0,C 180,E1 -12171.76,E2 -12171.76} C_VEL
LIN {X 0,Y 387.614,Z 409.618,A -85,B 0,C 180,E1 -12172.32,E2 -12172.32} C_VEL
LIN {X 0,Y 382.742,Z 401.882,A -85,B 0,C 180,E1 -12173.006,E2 -12173.006} C_VEL
LIN {X 0,Y 380.629,Z 396.677,A -85,B 0,C 180,E1 -12173.358,E2 -12173.358} C_VEL
LIN {X 0,Y 376.187,Z 383.534,A -85,B 0,C 180,E1 -12174.07,E2 -12174.07} C_VEL
LIN {X 0,Y 375.61,Z 381.24,A -85,B 0,C 180,E1 -12174.194,E2 -12174.194} C_VEL
LIN {X 0,Y 375.787,Z 377.514,A -85,B 0,C 180,E1 -12176.67,E2 -12176.67} C_VEL
LIN {X 0,Y 376.109,Z 372.338,A -85,B 0,C 180,E1 -12180.3,E2 -12180.3} C_VEL
LIN {X 0,Y 376.444,Z 367.189,A -85,B 0,C 180,E1 -12184.062,E2 -12184.062} C_VEL
LIN {X 0,Y 376.73,Z 363.763,A -85,B 0,C 180,E1 -12186.661,E2 -12186.661} C_VEL
LIN {X 0,Y 376.782,Z 360.324,A -85,B 0,C 180,E1 -12189.361,E2 -12189.361} C_VEL
LIN {X 0,Y 376.389,Z 356.824,A -85,B 0,C 180,E1 -12192.238,E2 -12192.238} C_VEL
LIN {X 0,Y 375.958,Z 354.281,A -85,B 0,C 180,E1 -12194.482,E2 -12194.482} C_VEL
LIN {X 0,Y 375.935,Z 354.279,A -85,B 0,C 180,E1 -12197.7,E2 -12197.7} C_VEL
LIN {X 0,Y 375.966,Z 354.275,A -85,B 0,C 180,E1 -12200.538,E2 -12200.538} C_VEL
LIN {X 0,Y 375.968,Z 354.278,A -85,B 0,C 180,E1 -12203.496,E2 -12203.496} C_VEL
LIN {X 0,Y 375.964,Z 354.277,A -85,B 0,C 180,E1 -12205.889,E2 -12205.889} C_VEL
LIN {X 0,Y 375.969,Z 354.278,A -85,B 0,C 180,E1 -12209.688,E2 -12209.688} C_VEL
LIN {X 0,Y 376.001,Z 354.274,A -85,B 0,C 180,E1 -12212.141,E2 -12212.141} C_VEL
LIN {X 0,Y 376.011,Z 354.271,A -85,B 0,C 180,E1 -12214.539,E2 -12214.539} C_VEL
LIN {X 0,Y 375.968,Z 354.28,A -85,B 0,C 180,E1 -12218.046,E2 -12218.046} C_VEL
LIN {X 0,Y 376.014,Z 354.272,A -85,B 0,C 180,E1 -12221.473,E2 -12221.473} C_VEL
LIN {X 0,Y 376.064,Z 354.264,A -85,B 0,C 180,E1 -12224.833,E2 -12224.833} C_VEL
LIN {X 0,Y 376.055,Z 354.264,A -85,B 0,C 180,E1 -12228.137,E2 -12228.137} C_VEL
LIN {X 0,Y 376.263,Z 354.239,A -85,B 0,C 180,E1 -12231.877,E2 -12231.877} C_VEL
LIN {X 0,Y 376.177,Z 354.249,A -85,B 0,C 180,E1 -12234.64,E2 -12234.64} C_VEL
LIN {X 0,Y 376.357,Z 354.227,A -85,B 0,C 180,E1 -12237.859,E2 -12237.859} C_VEL
LIN {X 0,Y 376.493,Z 354.215,A -85,B 0,C 180,E1 -12240,E2 -12240} C_VEL
LIN {X 0,Y 376.189,Z 354.251,A -85,B 0,C 180,E1 -12243.213,E2 -12243.213} C_VEL
LIN {X 0,Y 376.234,Z 354.246,A -85,B 0,C 180,E1 -12246.435,E2 -12246.435} C_VEL
LIN {X 0,Y 376.12,Z 354.261,A -85,B 0,C 180,E1 -12249.681,E2 -12249.681} C_VEL
LIN {X 0,Y 376.094,Z 354.263,A -85,B 0,C 180,E1 -12253.658,E2 -12253.658} C_VEL
LIN {X 0,Y 376.049,Z 354.271,A -85,B 0,C 180,E1 -12257.607,E2 -12257.607} C_VEL
LIN {X 0,Y 375.982,Z 354.28,A -85,B 0,C 180,E1 -12260.832,E2 -12260.832} C_VEL
LIN {X 0,Y 375.998,Z 354.276,A -85,B 0,C 180,E1 -12264.281,E2 -12264.281} C_VEL
LIN {X 0,Y 376.023,Z 354.273,A -85,B 0,C 180,E1 -12266.652,E2 -12266.652} C_VEL
LIN {X 0,Y 375.974,Z 354.278,A -85,B 0,C 180,E1 -12269.079,E2 -12269.079} C_VEL
LIN {X 0,Y 375.954,Z 354.283,A -85,B 0,C 180,E1 -12272.828,E2 -12272.828} C_VEL
LIN {X 0,Y 375.961,Z 354.284,A -85,B 0,C 180,E1 -12275.415,E2 -12275.415} C_VEL
LIN {X 0,Y 375.978,Z 354.279,A -85,B 0,C 180,E1 -12278.27,E2 -12278.27} C_VEL
LIN {X 0,Y 375.936,Z 354.284,A -85,B 0,C 180,E1 -12281.6,E2 -12281.6} C_VEL
LIN {X 0,Y 375.991,Z 354.446,A -85,B 0,C 180,E1 -12282.536,E2 -12282.536} C_VEL
LIN {X 0,Y 377.105,Z 359.882,A -85,B 0,C 180,E1 -12285.775,E2 -12285.775} C_VEL
LIN {X 0,Y 378.096,Z 365.262,A -85,B 0,C 180,E1 -12288.761,E2 -12288.761} C_VEL
LIN {X 0,Y 379.241,Z 370.99,A -85,B 0,C 180,E1 -12291.745,E2 -12291.745} C_VEL
LIN {X 0,Y 379.779,Z 374.939,A -85,B 0,C 180,E1 -12293.688,E2 -12293.688} C_VEL
LIN {X 0,Y 379.409,Z 379.169,A -85,B 0,C 180,E1 -12295.599,E2 -12295.599} C_VEL
LIN {X 0,Y 378.274,Z 387.531,A -85,B 0,C 180,E1 -12299.278,E2 -12299.278} C_VEL
LIN {X 0,Y 377.207,Z 396.458,A -85,B 0,C 180,E1 -12303.136,E2 -12303.136} C_VEL
LIN {X 0,Y 377.201,Z 397.082,A -85,B 0,C 180,E1 -12303.304,E2 -12303.304} C_VEL
LIN {X 0,Y 381.389,Z 413.391,A -85,B 0,C 180,E1 -12304.052,E2 -12304.052} C_VEL
LIN {X 0,Y 384.243,Z 427.656,A -85,B 0,C 180,E1 -12304.855,E2 -12304.855} C_VEL
LIN {X 0,Y 385.806,Z 438.395,A -85,B 0,C 180,E1 -12305.55,E2 -12305.55} C_VEL
LIN {X 0,Y 384.645,Z 452.251,A -85,B 0,C 180,E1 -12306.441,E2 -12306.441} C_VEL
LIN {X 0,Y 383.229,Z 465.389,A -85,B 0,C 180,E1 -12307.491,E2 -12307.491} C_VEL
LIN {X 0,Y 381.553,Z 478.783,A -85,B 0,C 180,E1 -12308.808,E2 -12308.808} C_VEL
LIN {X 0,Y 380.042,Z 491.013,A -85,B 0,C 180,E1 -12310.276,E2 -12310.276} C_VEL
LIN {X 0,Y 378.7,Z 502.204,A -85,B 0,C 180,E1 -12311.889,E2 -12311.889} C_VEL
LIN {X 0,Y 377.479,Z 511.669,A -85,B 0,C 180,E1 -12313.505,E2 -12313.505} C_VEL
LIN {X 0,Y 376.45,Z 520.966,A -85,B 0,C 180,E1 -12315.402,E2 -12315.402} C_VEL
LIN {X 0,Y 375.561,Z 529.702,A -85,B 0,C 180,E1 -12317.572,E2 -12317.572} C_VEL
LIN {X 0,Y 374.959,Z 536.706,A -85,B 0,C 180,E1 -12319.743,E2 -12319.743} C_VEL
LIN {X 0,Y 374.708,Z 542.211,A -85,B 0,C 180,E1 -12321.913,E2 -12321.913} C_VEL
LIN {X 0,Y 374.575,Z 546.085,A -85,B 0,C 180,E1 -12323.941,E2 -12323.941} C_VEL
LIN {X 0,Y 374.545,Z 548.514,A -85,B 0,C 180,E1 -12325.695,E2 -12325.695} C_VEL
LIN {X 0,Y 374.578,Z 550.388,A -85,B 0,C 180,E1 -12327.849,E2 -12327.849} C_VEL
LIN {X 0,Y 374.604,Z 551.026,A -85,B 0,C 180,E1 -12330,E2 -12330} C_VEL
LIN {X 0,Y 374.578,Z 550.382,A -85,B 0,C 180,E1 -12332.15,E2 -12332.15} C_VEL
LIN {X 0,Y 374.549,Z 548.502,A -85,B 0,C 180,E1 -12334.304,E2 -12334.304} C_VEL
LIN {X 0,Y 374.622,Z 545.371,A -85,B 0,C 180,E1 -12336.463,E2 -12336.463} C_VEL
LIN {X 0,Y 374.745,Z 540.92,A -85,B 0,C 180,E1 -12338.629,E2 -12338.629} C_VEL
LIN {X 0,Y 375.096,Z 535.05,A -85,B 0,C 180,E1 -12340.799,E2 -12340.799} C_VEL
LIN {X 0,Y 375.656,Z 528.655,A -85,B 0,C 180,E1 -12342.699,E2 -12342.699} C_VEL
LIN {X 0,Y 376.45,Z 520.927,A -85,B 0,C 180,E1 -12344.598,E2 -12344.598} C_VEL
LIN {X 0,Y 377.475,Z 511.626,A -85,B 0,C 180,E1 -12346.495,E2 -12346.495} C_VEL
LIN {X 0,Y 378.669,Z 502.153,A -85,B 0,C 180,E1 -12348.112,E2 -12348.112} C_VEL
LIN {X 0,Y 380.053,Z 490.958,A -85,B 0,C 180,E1 -12349.724,E2 -12349.724} C_VEL
LIN {X 0,Y 381.557,Z 478.719,A -85,B 0,C 180,E1 -12351.191,E2 -12351.191} C_VEL
LIN {X 0,Y 383.146,Z 465.288,A -85,B 0,C 180,E1 -12352.514,E2 -12352.514} C_VEL
LIN {X 0,Y 384.663,Z 452.13,A -85,B 0,C 180,E1 -12353.557,E2 -12353.557} C_VEL
LIN {X 0,Y 385.767,Z 437.831,A -85,B 0,C 180,E1 -12354.479,E2 -12354.479} C_VEL
LIN {X 0,Y 383.45,Z 423.254,A -85,B 0,C 180,E1 -12355.4,E2 -12355.4} C_VEL
LIN {X 0,Y 380.126,Z 408.099,A -85,B 0,C 180,E1 -12356.199,E2 -12356.199} C_VEL
LIN {X 0,Y 377.178,Z 396.778,A -85,B 0,C 180,E1 -12356.712,E2 -12356.712} C_VEL
LIN {X 0,Y 378.078,Z 388.896,A -85,B 0,C 180,E1 -12360.126,E2 -12360.126} C_VEL
LIN {X 0,Y 379.203,Z 380.545,A -85,B 0,C 180,E1 -12363.78,E2 -12363.78} C_VEL
LIN {X 0,Y 379.717,Z 376.717,A -85,B 0,C 180,E1 -12365.475,E2 -12365.475} C_VEL
LIN {X 0,Y 379.558,Z 372.99,A -85,B 0,C 180,E1 -12367.232,E2 -12367.232} C_VEL
LIN {X 0,Y 378.322,Z 366.483,A -85,B 0,C 180,E1 -12370.556,E2 -12370.556} C_VEL
LIN {X 0,Y 377.311,Z 360.971,A -85,B 0,C 180,E1 -12373.566,E2 -12373.566} C_VEL
LIN {X 0,Y 375.972,Z 354.278,A -85,B 0,C 180,E1 -12377.553,E2 -12377.553} C_VEL
LIN {X 0,Y 375.971,Z 354.28,A -85,B 0,C 180,E1 -12380.539,E2 -12380.539} C_VEL
LIN {X 0,Y 375.967,Z 354.283,A -85,B 0,C 180,E1 -12383.495,E2 -12383.495} C_VEL
LIN {X 0,Y 375.964,Z 354.283,A -85,B 0,C 180,E1 -12385.889,E2 -12385.889} C_VEL
LIN {X 0,Y 375.967,Z 354.282,A -85,B 0,C 180,E1 -12389.688,E2 -12389.688} C_VEL
LIN {X 0,Y 375.998,Z 354.274,A -85,B 0,C 180,E1 -12392.142,E2 -12392.142} C_VEL
LIN {X 0,Y 376.009,Z 354.273,A -85,B 0,C 180,E1 -12394.539,E2 -12394.539} C_VEL
LIN {X 0,Y 375.966,Z 354.279,A -85,B 0,C 180,E1 -12398.046,E2 -12398.046} C_VEL
LIN {X 0,Y 376.027,Z 354.268,A -85,B 0,C 180,E1 -12401.474,E2 -12401.474} C_VEL
LIN {X 0,Y 376.063,Z 354.264,A -85,B 0,C 180,E1 -12404.833,E2 -12404.833} C_VEL
LIN {X 0,Y 376.062,Z 354.266,A -85,B 0,C 180,E1 -12408.137,E2 -12408.137} C_VEL
LIN {X 0,Y 376.204,Z 354.249,A -85,B 0,C 180,E1 -12411.938,E2 -12411.938} C_VEL
LIN {X 0,Y 376.172,Z 354.251,A -85,B 0,C 180,E1 -12414.64,E2 -12414.64} C_VEL
LIN {X 0,Y 376.356,Z 354.226,A -85,B 0,C 180,E1 -12417.86,E2 -12417.86} C_VEL
LIN {X 0,Y 376.491,Z 354.209,A -85,B 0,C 180,E1 -12420,E2 -12420} C_VEL
LIN {X 0,Y 376.188,Z 354.25,A -85,B 0,C 180,E1 -12423.213,E2 -12423.213} C_VEL
LIN {X 0,Y 376.238,Z 354.244,A -85,B 0,C 180,E1 -12426.64,E2 -12426.64} C_VEL
LIN {X 0,Y 376.21,Z 354.246,A -85,B 0,C 180,E1 -12428.595,E2 -12428.595} C_VEL
LIN {X 0,Y 376.062,Z 354.263,A -85,B 0,C 180,E1 -12431.863,E2 -12431.863} C_VEL
LIN {X 0,Y 376.064,Z 354.263,A -85,B 0,C 180,E1 -12435.167,E2 -12435.167} C_VEL
LIN {X 0,Y 376.028,Z 354.268,A -85,B 0,C 180,E1 -12438.526,E2 -12438.526} C_VEL
LIN {X 0,Y 375.967,Z 354.278,A -85,B 0,C 180,E1 -12441.954,E2 -12441.954} C_VEL
LIN {X 0,Y 376.01,Z 354.273,A -85,B 0,C 180,E1 -12445.461,E2 -12445.461} C_VEL
LIN {X 0,Y 375.974,Z 354.274,A -85,B 0,C 180,E1 -12449.079,E2 -12449.079} C_VEL
LIN {X 0,Y 375.952,Z 354.279,A -85,B 0,C 180,E1 -12452.828,E2 -12452.828} C_VEL
LIN {X 0,Y 375.96,Z 354.281,A -85,B 0,C 180,E1 -12455.415,E2 -12455.415} C_VEL
LIN {X 0,Y 375.977,Z 354.277,A -85,B 0,C 180,E1 -12458.27,E2 -12458.27} C_VEL
LIN {X 0,Y 375.937,Z 354.283,A -85,B 0,C 180,E1 -12461.601,E2 -12461.601} C_VEL
LIN {X 0,Y 375.929,Z 354.286,A -85,B 0,C 180,E1 -12465.269,E2 -12465.269} C_VEL
LIN {X 0,Y 375.976,Z 354.367,A -85,B 0,C 180,E1 -12465.766,E2 -12465.766} C_VEL
LIN {X 0,Y 376.61,Z 358.428,A -85,B 0,C 180,E1 -12469.221,E2 -12469.221} C_VEL
LIN {X 0,Y 376.778,Z 361.884,A -85,B 0,C 180,E1 -12472.008,E2 -12472.008} C_VEL
LIN {X 0,Y 376.54,Z 366.047,A -85,B 0,C 180,E1 -12475.21,E2 -12475.21} C_VEL
LIN {X 0,Y 376.198,Z 370.44,A -85,B 0,C 180,E1 -12478.46,E2 -12478.46} C_VEL
LIN {X 0,Y 375.872,Z 375.622,A -85,B 0,C 180,E1 -12482.131,E2 -12482.131} C_VEL
LIN {X 0,Y 375.714,Z 379.139,A -85,B 0,C 180,E1 -12484.518,E2 -12484.518} C_VEL
LIN {X 0,Y 375.617,Z 381.259,A -85,B 0,C 180,E1 -12485.918,E2 -12485.918} C_VEL
LIN {X 0,Y 380.949,Z 397.9,A -85,B 0,C 180,E1 -12486.812,E2 -12486.812} C_VEL
LIN {X 0,Y 384.327,Z 410.738,A -85,B 0,C 180,E1 -12487.633,E2 -12487.633} C_VEL
LIN {X 0,Y 385.775,Z 417.292,A -85,B 0,C 180,E1 -12488.106,E2 -12488.106} C_VEL
LIN {X 0,Y 385.032,Z 429.32,A -85,B 0,C 180,E1 -12488.893,E2 -12488.893} C_VEL
LIN {X 0,Y 383.714,Z 441.962,A -85,B 0,C 180,E1 -12489.915,E2 -12489.915} C_VEL
LIN {X 0,Y 382.316,Z 453.676,A -85,B 0,C 180,E1 -12491.095,E2 -12491.095} C_VEL
LIN {X 0,Y 380.915,Z 465.327,A -85,B 0,C 180,E1 -12492.553,E2 -12492.553} C_VEL
LIN {X 0,Y 379.384,Z 476.187,A -85,B 0,C 180,E1 -12494.222,E2 -12494.222} C_VEL
LIN {X 0,Y 378.141,Z 485.6,A -85,B 0,C 180,E1 -12496.018,E2 -12496.018} C_VEL
LIN {X 0,Y 377.003,Z 493.537,A -85,B 0,C 180,E1 -12497.894,E2 -12497.894} C_VEL
LIN {X 0,Y 376.151,Z 499.94,A -85,B 0,C 180,E1 -12499.776,E2 -12499.776} C_VEL
LIN {X 0,Y 375.442,Z 505.626,A -85,B 0,C 180,E1 -12501.929,E2 -12501.929} C_VEL
LIN {X 0,Y 375.151,Z 508.907,A -85,B 0,C 180,E1 -12503.546,E2 -12503.546} C_VEL
LIN {X 0,Y 374.765,Z 512.062,A -85,B 0,C 180,E1 -12505.698,E2 -12505.698} C_VEL
LIN {X 0,Y 374.746,Z 513.913,A -85,B 0,C 180,E1 -12507.851,E2 -12507.851} C_VEL
LIN {X 0,Y 374.608,Z 514.548,A -85,B 0,C 180,E1 -12510,E2 -12510} C_VEL
LIN {X 0,Y 374.745,Z 513.971,A -85,B 0,C 180,E1 -12512.15,E2 -12512.15} C_VEL
LIN {X 0,Y 374.763,Z 512.183,A -85,B 0,C 180,E1 -12514.302,E2 -12514.302} C_VEL
LIN {X 0,Y 375.148,Z 509.09,A -85,B 0,C 180,E1 -12516.454,E2 -12516.454} C_VEL
LIN {X 0,Y 375.56,Z 504.6,A -85,B 0,C 180,E1 -12518.61,E2 -12518.61} C_VEL
LIN {X 0,Y 376.32,Z 498.552,A -85,B 0,C 180,E1 -12520.764,E2 -12520.764} C_VEL
LIN {X 0,Y 377.212,Z 491.811,A -85,B 0,C 180,E1 -12522.646,E2 -12522.646} C_VEL
LIN {X 0,Y 378.488,Z 483.438,A -85,B 0,C 180,E1 -12524.518,E2 -12524.518} C_VEL
LIN {X 0,Y 379.581,Z 474.702,A -85,B 0,C 180,E1 -12526.125,E2 -12526.125} C_VEL
LIN {X 0,Y 381.098,Z 464.084,A -85,B 0,C 180,E1 -12527.715,E2 -12527.715} C_VEL
LIN {X 0,Y 382.453,Z 453.331,A -85,B 0,C 180,E1 -12529.037,E2 -12529.037} C_VEL
LIN {X 0,Y 383.789,Z 441.552,A -85,B 0,C 180,E1 -12530.221,E2 -12530.221} C_VEL
LIN {X 0,Y 385.089,Z 428.545,A -85,B 0,C 180,E1 -12531.266,E2 -12531.266} C_VEL
LIN {X 0,Y 385.875,Z 418.201,A -85,B 0,C 180,E1 -12531.932,E2 -12531.932} C_VEL
LIN {X 0,Y 383.209,Z 406.038,A -85,B 0,C 180,E1 -12532.783,E2 -12532.783} C_VEL
LIN {X 0,Y 380.629,Z 396.677,A -85,B 0,C 180,E1 -12533.358,E2 -12533.358} C_VEL
LIN {X 0,Y 379.478,Z 395.103,A -85,B 0,C 180,E1 -12533.5,E2 -12533.5} C_VEL
LIN {X 0,Y 372.808,Z 392.346,A -85,B 0,C 180,E1 -12534.074,E2 -12534.074} C_VEL
LIN {X 0,Y 371.799,Z 390.997,A -85,B 0,C 180,E1 -12534.191,E2 -12534.191} C_VEL
LIN {X 0,Y 368.687,Z 382.029,A -85,B 0,C 180,E1 -12534.665,E2 -12534.665} C_VEL
LIN {X 0,Y 368.598,Z 381.382,A -85,B 0,C 180,E1 -12534.729,E2 -12534.729} C_VEL
LIN {X 0,Y 368.783,Z 377.724,A -85,B 0,C 180,E1 -12537.218,E2 -12537.218} C_VEL
LIN {X 0,Y 369.137,Z 372.371,A -85,B 0,C 180,E1 -12541.045,E2 -12541.045} C_VEL
LIN {X 0,Y 369.511,Z 367.353,A -85,B 0,C 180,E1 -12544.792,E2 -12544.792} C_VEL
LIN {X 0,Y 369.761,Z 363.918,A -85,B 0,C 180,E1 -12547.461,E2 -12547.461} C_VEL
LIN {X 0,Y 369.723,Z 360.461,A -85,B 0,C 180,E1 -12550.264,E2 -12550.264} C_VEL
LIN {X 0,Y 369.181,Z 356.474,A -85,B 0,C 180,E1 -12553.664,E2 -12553.664} C_VEL
LIN {X 0,Y 368.893,Z 355.16,A -85,B 0,C 180,E1 -12555.002,E2 -12555.002} C_VEL
LIN {X 0,Y 368.887,Z 355.157,A -85,B 0,C 180,E1 -12558.178,E2 -12558.178} C_VEL
LIN {X 0,Y 368.912,Z 355.156,A -85,B 0,C 180,E1 -12561.36,E2 -12561.36} C_VEL
LIN {X 0,Y 368.941,Z 355.154,A -85,B 0,C 180,E1 -12565.147,E2 -12565.147} C_VEL
LIN {X 0,Y 368.933,Z 355.154,A -85,B 0,C 180,E1 -12569.047,E2 -12569.047} C_VEL
LIN {X 0,Y 368.984,Z 355.148,A -85,B 0,C 180,E1 -12571.564,E2 -12571.564} C_VEL
LIN {X 0,Y 369.005,Z 355.142,A -85,B 0,C 180,E1 -12574.02,E2 -12574.02} C_VEL
LIN {X 0,Y 368.937,Z 355.153,A -85,B 0,C 180,E1 -12577.605,E2 -12577.605} C_VEL
LIN {X 0,Y 368.963,Z 355.151,A -85,B 0,C 180,E1 -12581.106,E2 -12581.106} C_VEL
LIN {X 0,Y 369.003,Z 355.145,A -85,B 0,C 180,E1 -12584.535,E2 -12584.535} C_VEL
LIN {X 0,Y 369.01,Z 355.142,A -85,B 0,C 180,E1 -12587.907,E2 -12587.907} C_VEL
LIN {X 0,Y 369.235,Z 355.114,A -85,B 0,C 180,E1 -12591.8,E2 -12591.8} C_VEL
LIN {X 0,Y 369.15,Z 355.124,A -85,B 0,C 180,E1 -12594.537,E2 -12594.537} C_VEL
LIN {X 0,Y 369.322,Z 355.103,A -85,B 0,C 180,E1 -12597.819,E2 -12597.819} C_VEL
LIN {X 0,Y 369.462,Z 355.091,A -85,B 0,C 180,E1 -12600,E2 -12600} C_VEL
LIN {X 0,Y 369.322,Z 355.105,A -85,B 0,C 180,E1 -12602.181,E2 -12602.181} C_VEL
LIN {X 0,Y 369.193,Z 355.124,A -85,B 0,C 180,E1 -12606.558,E2 -12606.558} C_VEL
LIN {X 0,Y 369.07,Z 355.14,A -85,B 0,C 180,E1 -12609.868,E2 -12609.868} C_VEL
LIN {X 0,Y 369.042,Z 355.141,A -85,B 0,C 180,E1 -12613.772,E2 -12613.772} C_VEL
LIN {X 0,Y 369.005,Z 355.148,A -85,B 0,C 180,E1 -12617.768,E2 -12617.768} C_VEL
LIN {X 0,Y 368.933,Z 355.158,A -85,B 0,C 180,E1 -12621.219,E2 -12621.219} C_VEL
LIN {X 0,Y 368.962,Z 355.152,A -85,B 0,C 180,E1 -12624.775,E2 -12624.775} C_VEL
LIN {X 0,Y 368.972,Z 355.152,A -85,B 0,C 180,E1 -12627.203,E2 -12627.203} C_VEL
LIN {X 0,Y 368.922,Z 355.154,A -85,B 0,C 180,E1 -12629.689,E2 -12629.689} C_VEL
LIN {X 0,Y 368.901,Z 355.162,A -85,B 0,C 180,E1 -12633.043,E2 -12633.043} C_VEL
LIN {X 0,Y 368.921,Z 355.16,A -85,B 0,C 180,E1 -12636.196,E2 -12636.196} C_VEL
LIN {X 0,Y 368.907,Z 355.16,A -85,B 0,C 180,E1 -12638.953,E2 -12638.953} C_VEL
LIN {X 0,Y 368.895,Z 355.201,A -85,B 0,C 180,E1 -12641.821,E2 -12641.821} C_VEL
LIN {X 0,Y 369.851,Z 359.782,A -85,B 0,C 180,E1 -12644.675,E2 -12644.675} C_VEL
LIN {X 0,Y 370.85,Z 364.916,A -85,B 0,C 180,E1 -12647.654,E2 -12647.654} C_VEL
LIN {X 0,Y 372.197,Z 372,A -85,B 0,C 180,E1 -12651.455,E2 -12651.455} C_VEL
LIN {X 0,Y 372.816,Z 376.191,A -85,B 0,C 180,E1 -12653.572,E2 -12653.572} C_VEL
LIN {X 0,Y 372.439,Z 380.387,A -85,B 0,C 180,E1 -12655.52,E2 -12655.52} C_VEL
LIN {X 0,Y 371.271,Z 388.702,A -85,B 0,C 180,E1 -12659.263,E2 -12659.263} C_VEL
LIN {X 0,Y 370.229,Z 396.626,A -85,B 0,C 180,E1 -12662.776,E2 -12662.776} C_VEL
LIN {X 0,Y 374.741,Z 413.991,A -85,B 0,C 180,E1 -12663.612,E2 -12663.612} C_VEL
LIN {X 0,Y 377.671,Z 429.074,A -85,B 0,C 180,E1 -12664.493,E2 -12664.493} C_VEL
LIN {X 0,Y 379.192,Z 440.209,A -85,B 0,C 180,E1 -12665.254,E2 -12665.254} C_VEL
LIN {X 0,Y 377.9,Z 453.47,A -85,B 0,C 180,E1 -12666.14,E2 -12666.14} C_VEL
LIN {X 0,Y 376.438,Z 466.331,A -85,B 0,C 180,E1 -12667.207,E2 -12667.207} C_VEL
LIN {X 0,Y 374.729,Z 479.518,A -85,B 0,C 180,E1 -12668.548,E2 -12668.548} C_VEL
LIN {X 0,Y 373.229,Z 490.592,A -85,B 0,C 180,E1 -12669.9,E2 -12669.9} C_VEL
LIN {X 0,Y 371.881,Z 501.806,A -85,B 0,C 180,E1 -12671.545,E2 -12671.545} C_VEL
LIN {X 0,Y 370.559,Z 511.276,A -85,B 0,C 180,E1 -12673.188,E2 -12673.188} C_VEL
LIN {X 0,Y 369.475,Z 520.586,A -85,B 0,C 180,E1 -12675.12,E2 -12675.12} C_VEL
LIN {X 0,Y 368.563,Z 529.337,A -85,B 0,C 180,E1 -12677.332,E2 -12677.332} C_VEL
LIN {X 0,Y 367.915,Z 536.348,A -85,B 0,C 180,E1 -12679.544,E2 -12679.544} C_VEL
LIN {X 0,Y 367.62,Z 541.857,A -85,B 0,C 180,E1 -12681.756,E2 -12681.756} C_VEL
LIN {X 0,Y 367.494,Z 545.969,A -85,B 0,C 180,E1 -12683.962,E2 -12683.962} C_VEL
LIN {X 0,Y 367.471,Z 548.167,A -85,B 0,C 180,E1 -12685.612,E2 -12685.612} C_VEL
LIN {X 0,Y 367.478,Z 550.042,A -85,B 0,C 180,E1 -12687.808,E2 -12687.808} C_VEL
LIN {X 0,Y 367.538,Z 550.681,A -85,B 0,C 180,E1 -12690,E2 -12690} C_VEL
LIN {X 0,Y 367.478,Z 550.036,A -85,B 0,C 180,E1 -12692.192,E2 -12692.192} C_VEL
LIN {X 0,Y 367.476,Z 548.155,A -85,B 0,C 180,E1 -12694.387,E2 -12694.387} C_VEL
LIN {X 0,Y 367.549,Z 545.019,A -85,B 0,C 180,E1 -12696.588,E2 -12696.588} C_VEL
LIN {X 0,Y 367.688,Z 540.563,A -85,B 0,C 180,E1 -12698.796,E2 -12698.796} C_VEL
LIN {X 0,Y 368.075,Z 534.687,A -85,B 0,C 180,E1 -12701.008,E2 -12701.008} C_VEL
LIN {X 0,Y 368.646,Z 527.24,A -85,B 0,C 180,E1 -12703.225,E2 -12703.225} C_VEL
LIN {X 0,Y 369.617,Z 519.284,A -85,B 0,C 180,E1 -12705.156,E2 -12705.156} C_VEL
LIN {X 0,Y 370.733,Z 509.716,A -85,B 0,C 180,E1 -12707.088,E2 -12707.088} C_VEL
LIN {X 0,Y 372.023,Z 499.987,A -85,B 0,C 180,E1 -12708.733,E2 -12708.733} C_VEL
LIN {X 0,Y 373.549,Z 488.439,A -85,B 0,C 180,E1 -12710.369,E2 -12710.369} C_VEL
LIN {X 0,Y 375.173,Z 475.738,A -85,B 0,C 180,E1 -12711.858,E2 -12711.858} C_VEL
LIN {X 0,Y 376.724,Z 463.241,A -85,B 0,C 180,E1 -12713.065,E2 -12713.065} C_VEL
LIN {X 0,Y 378.409,Z 448.691,A -85,B 0,C 180,E1 -12714.191,E2 -12714.191} C_VEL
LIN {X 0,Y 379.151,Z 439.285,A -85,B 0,C 180,E1 -12714.799,E2 -12714.799} C_VEL
LIN {X 0,Y 376.872,Z 424.484,A -85,B 0,C 180,E1 -12715.777,E2 -12715.777} C_VEL
LIN {X 0,Y 373.619,Z 409.471,A -85,B 0,C 180,E1 -12716.609,E2 -12716.609} C_VEL
LIN {X 0,Y 370.281,Z 396.554,A -85,B 0,C 180,E1 -12717.236,E2 -12717.236} C_VEL
LIN {X 0,Y 371.414,Z 387.647,A -85,B 0,C 180,E1 -12721.197,E2 -12721.197} C_VEL
LIN {X 0,Y 372.609,Z 378.964,A -85,B 0,C 180,E1 -12725.119,E2 -12725.119} C_VEL
LIN {X 0,Y 372.805,Z 376.139,A -85,B 0,C 180,E1 -12726.429,E2 -12726.429} C_VEL
LIN {X 0,Y 372.18,Z 371.912,A -85,B 0,C 180,E1 -12728.547,E2 -12728.547} C_VEL
LIN {X 0,Y 370.823,Z 364.876,A -85,B 0,C 180,E1 -12732.342,E2 -12732.342} C_VEL
LIN {X 0,Y 369.825,Z 359.723,A -85,B 0,C 180,E1 -12735.321,E2 -12735.321} C_VEL
LIN {X 0,Y 368.917,Z 355.148,A -85,B 0,C 180,E1 -12738.183,E2 -12738.183} C_VEL
LIN {X 0,Y 368.915,Z 355.16,A -85,B 0,C 180,E1 -12741.359,E2 -12741.359} C_VEL
LIN {X 0,Y 368.939,Z 355.159,A -85,B 0,C 180,E1 -12745.147,E2 -12745.147} C_VEL
LIN {X 0,Y 368.931,Z 355.159,A -85,B 0,C 180,E1 -12749.047,E2 -12749.047} C_VEL
LIN {X 0,Y 368.982,Z 355.151,A -85,B 0,C 180,E1 -12751.564,E2 -12751.564} C_VEL
LIN {X 0,Y 369.002,Z 355.146,A -85,B 0,C 180,E1 -12754.02,E2 -12754.02} C_VEL
LIN {X 0,Y 368.935,Z 355.154,A -85,B 0,C 180,E1 -12757.605,E2 -12757.605} C_VEL
LIN {X 0,Y 368.986,Z 355.146,A -85,B 0,C 180,E1 -12761.108,E2 -12761.108} C_VEL
LIN {X 0,Y 369.002,Z 355.141,A -85,B 0,C 180,E1 -12764.536,E2 -12764.536} C_VEL
LIN {X 0,Y 369.016,Z 355.141,A -85,B 0,C 180,E1 -12767.907,E2 -12767.907} C_VEL
LIN {X 0,Y 369.151,Z 355.128,A -85,B 0,C 180,E1 -12771.889,E2 -12771.889} C_VEL
LIN {X 0,Y 369.144,Z 355.126,A -85,B 0,C 180,E1 -12774.538,E2 -12774.538} C_VEL
LIN {X 0,Y 369.32,Z 355.102,A -85,B 0,C 180,E1 -12777.819,E2 -12777.819} C_VEL
LIN {X 0,Y 369.461,Z 355.084,A -85,B 0,C 180,E1 -12780,E2 -12780} C_VEL
LIN {X 0,Y 369.32,Z 355.106,A -85,B 0,C 180,E1 -12782.181,E2 -12782.181} C_VEL
LIN {X 0,Y 369.207,Z 355.12,A -85,B 0,C 180,E1 -12786.628,E2 -12786.628} C_VEL
LIN {X 0,Y 369.143,Z 355.128,A -85,B 0,C 180,E1 -12788.761,E2 -12788.761} C_VEL
LIN {X 0,Y 369.017,Z 355.142,A -85,B 0,C 180,E1 -12792.093,E2 -12792.093} C_VEL
LIN {X 0,Y 369.003,Z 355.144,A -85,B 0,C 180,E1 -12795.465,E2 -12795.465} C_VEL
LIN {X 0,Y 368.986,Z 355.148,A -85,B 0,C 180,E1 -12798.893,E2 -12798.893} C_VEL
LIN {X 0,Y 368.936,Z 355.154,A -85,B 0,C 180,E1 -12802.395,E2 -12802.395} C_VEL
LIN {X 0,Y 369.004,Z 355.145,A -85,B 0,C 180,E1 -12805.98,E2 -12805.98} C_VEL
LIN {X 0,Y 368.964,Z 355.149,A -85,B 0,C 180,E1 -12808.812,E2 -12808.812} C_VEL
LIN {X 0,Y 368.901,Z 355.158,A -85,B 0,C 180,E1 -12812.238,E2 -12812.238} C_VEL
LIN {X 0,Y 368.932,Z 355.156,A -85,B 0,C 180,E1 -12815.002,E2 -12815.002} C_VEL
LIN {X 0,Y 368.911,Z 355.157,A -85,B 0,C 180,E1 -12818.64,E2 -12818.64} C_VEL
LIN {X 0,Y 368.884,Z 355.162,A -85,B 0,C 180,E1 -12822.009,E2 -12822.009} C_VEL
LIN {X 0,Y 368.937,Z 355.284,A -85,B 0,C 180,E1 -12825.401,E2 -12825.401} C_VEL
LIN {X 0,Y 369.476,Z 358.554,A -85,B 0,C 180,E1 -12828.26,E2 -12828.26} C_VEL
LIN {X 0,Y 369.778,Z 362.066,A -85,B 0,C 180,E1 -12831.192,E2 -12831.192} C_VEL
LIN {X 0,Y 369.623,Z 365.473,A -85,B 0,C 180,E1 -12833.883,E2 -12833.883} C_VEL
LIN {X 0,Y 369.357,Z 369.343,A -85,B 0,C 180,E1 -12836.848,E2 -12836.848} C_VEL
LIN {X 0,Y 368.984,Z 374.085,A -85,B 0,C 180,E1 -12840.316,E2 -12840.316} C_VEL
LIN {X 0,Y 368.731,Z 379.346,A -85,B 0,C 180,E1 -12843.999,E2 -12843.999} C_VEL
LIN {X 0,Y 368.596,Z 381.41,A -85,B 0,C 180,E1 -12845.392,E2 -12845.392} C_VEL
LIN {X 0,Y 374.322,Z 398.912,A -85,B 0,C 180,E1 -12846.38,E2 -12846.38} C_VEL
LIN {X 0,Y 377.718,Z 412.018,A -85,B 0,C 180,E1 -12847.251,E2 -12847.251} C_VEL
LIN {X 0,Y 379.262,Z 419.483,A -85,B 0,C 180,E1 -12847.808,E2 -12847.808} C_VEL
LIN {X 0,Y 378.205,Z 432.003,A -85,B 0,C 180,E1 -12848.664,E2 -12848.664} C_VEL
LIN {X 0,Y 376.918,Z 443.881,A -85,B 0,C 180,E1 -12849.679,E2 -12849.679} C_VEL
LIN {X 0,Y 375.493,Z 455.292,A -85,B 0,C 180,E1 -12850.88,E2 -12850.88} C_VEL
LIN {X 0,Y 374.162,Z 465.745,A -85,B 0,C 180,E1 -12852.228,E2 -12852.228} C_VEL
LIN {X 0,Y 372.617,Z 476.126,A -85,B 0,C 180,E1 -12853.847,E2 -12853.847} C_VEL
LIN {X 0,Y 371.441,Z 484.669,A -85,B 0,C 180,E1 -12855.481,E2 -12855.481} C_VEL
LIN {X 0,Y 370.19,Z 492.869,A -85,B 0,C 180,E1 -12857.389,E2 -12857.389} C_VEL
LIN {X 0,Y 369.398,Z 498.591,A -85,B 0,C 180,E1 -12859.032,E2 -12859.032} C_VEL
LIN {X 0,Y 368.557,Z 504.71,A -85,B 0,C 180,E1 -12861.225,E2 -12861.225} C_VEL
LIN {X 0,Y 368.084,Z 509.259,A -85,B 0,C 180,E1 -12863.422,E2 -12863.422} C_VEL
LIN {X 0,Y 367.696,Z 512.41,A -85,B 0,C 180,E1 -12865.615,E2 -12865.615} C_VEL
LIN {X 0,Y 367.666,Z 514.259,A -85,B 0,C 180,E1 -12867.809,E2 -12867.809} C_VEL
LIN {X 0,Y 367.542,Z 514.892,A -85,B 0,C 180,E1 -12870,E2 -12870} C_VEL
LIN {X 0,Y 367.665,Z 514.316,A -85,B 0,C 180,E1 -12872.191,E2 -12872.191} C_VEL
LIN {X 0,Y 367.695,Z 512.529,A -85,B 0,C 180,E1 -12874.385,E2 -12874.385} C_VEL
LIN {X 0,Y 368.082,Z 509.44,A -85,B 0,C 180,E1 -12876.579,E2 -12876.579} C_VEL
LIN {X 0,Y 368.546,Z 504.953,A -85,B 0,C 180,E1 -12878.775,E2 -12878.775} C_VEL
LIN {X 0,Y 369.345,Z 498.911,A -85,B 0,C 180,E1 -12880.969,E2 -12880.969} C_VEL
LIN {X 0,Y 370.294,Z 492.177,A -85,B 0,C 180,E1 -12882.886,E2 -12882.886} C_VEL
LIN {X 0,Y 371.623,Z 483.815,A -85,B 0,C 180,E1 -12884.792,E2 -12884.792} C_VEL
LIN {X 0,Y 372.769,Z 475.093,A -85,B 0,C 180,E1 -12886.428,E2 -12886.428} C_VEL
LIN {X 0,Y 374.346,Z 464.495,A -85,B 0,C 180,E1 -12888.046,E2 -12888.046} C_VEL
LIN {X 0,Y 375.783,Z 453.767,A -85,B 0,C 180,E1 -12889.388,E2 -12889.388} C_VEL
LIN {X 0,Y 377.165,Z 442.028,A -85,B 0,C 180,E1 -12890.592,E2 -12890.592} C_VEL
LIN {X 0,Y 378.459,Z 429.569,A -85,B 0,C 180,E1 -12891.618,E2 -12891.618} C_VEL
LIN {X 0,Y 379.206,Z 419.016,A -85,B 0,C 180,E1 -12892.327,E2 -12892.327} C_VEL
LIN {X 0,Y 376.212,Z 405.803,A -85,B 0,C 180,E1 -12893.28,E2 -12893.28} C_VEL
LIN {X 0,Y 372.149,Z 391.988,A -85,B 0,C 180,E1 -12894.134,E2 -12894.134} C_VEL
LIN {X 0,Y 371.799,Z 390.997,A -85,B 0,C 180,E1 -12894.191,E2 -12894.191} C_VEL
LIN {X 0,Y 369.961,Z 387.665,A -85,B 0,C 180,E1 -12894.456,E2 -12894.456} C_VEL
LIN {X 0,Y 367.535,Z 385.038,A -85,B 0,C 180,E1 -12894.806,E2 -12894.806} C_VEL
LIN {X 0,Y 364.299,Z 382.381,A -85,B 0,C 180,E1 -12895.391,E2 -12895.391} C_VEL
LIN {X 0,Y 362.231,Z 380.653,A -85,B 0,C 180,E1 -12896.023,E2 -12896.023} C_VEL
LIN {X 0,Y 361.721,Z 379.732,A -85,B 0,C 180,E1 -12896.535,E2 -12896.535} C_VEL
LIN {X 0,Y 362.032,Z 374.466,A -85,B 0,C 180,E1 -12900.314,E2 -12900.314} C_VEL
LIN {X 0,Y 362.434,Z 369.238,A -85,B 0,C 180,E1 -12904.218,E2 -12904.218} C_VEL
LIN {X 0,Y 362.762,Z 365.196,A -85,B 0,C 180,E1 -12907.409,E2 -12907.409} C_VEL
LIN {X 0,Y 362.739,Z 362.352,A -85,B 0,C 180,E1 -12909.745,E2 -12909.745} C_VEL
LIN {X 0,Y 362.363,Z 358.84,A -85,B 0,C 180,E1 -12912.752,E2 -12912.752} C_VEL
LIN {X 0,Y 361.839,Z 356.038,A -85,B 0,C 180,E1 -12915.305,E2 -12915.305} C_VEL
LIN {X 0,Y 361.831,Z 356.035,A -85,B 0,C 180,E1 -12918.67,E2 -12918.67} C_VEL
LIN {X 0,Y 361.872,Z 356.033,A -85,B 0,C 180,E1 -12921.575,E2 -12921.575} C_VEL
LIN {X 0,Y 361.878,Z 356.034,A -85,B 0,C 180,E1 -12924.655,E2 -12924.655} C_VEL
LIN {X 0,Y 361.842,Z 356.04,A -85,B 0,C 180,E1 -12928.371,E2 -12928.371} C_VEL
LIN {X 0,Y 361.904,Z 356.03,A -85,B 0,C 180,E1 -12930.955,E2 -12930.955} C_VEL
LIN {X 0,Y 361.959,Z 356.022,A -85,B 0,C 180,E1 -12933.475,E2 -12933.475} C_VEL
LIN {X 0,Y 361.895,Z 356.031,A -85,B 0,C 180,E1 -12937.145,E2 -12937.145} C_VEL
LIN {X 0,Y 361.912,Z 356.029,A -85,B 0,C 180,E1 -12940.723,E2 -12940.723} C_VEL
LIN {X 0,Y 361.938,Z 356.025,A -85,B 0,C 180,E1 -12943.066,E2 -12943.066} C_VEL
LIN {X 0,Y 362.004,Z 356.019,A -85,B 0,C 180,E1 -12946.528,E2 -12946.528} C_VEL
LIN {X 0,Y 362.036,Z 356.016,A -85,B 0,C 180,E1 -12949.938,E2 -12949.938} C_VEL
LIN {X 0,Y 362.157,Z 355.998,A -85,B 0,C 180,E1 -12952.192,E2 -12952.192} C_VEL
LIN {X 0,Y 362.123,Z 356,A -85,B 0,C 180,E1 -12954.431,E2 -12954.431} C_VEL
LIN {X 0,Y 362.286,Z 355.979,A -85,B 0,C 180,E1 -12957.776,E2 -12957.776} C_VEL
LIN {X 0,Y 362.432,Z 355.966,A -85,B 0,C 180,E1 -12960,E2 -12960} C_VEL
LIN {X 0,Y 362.286,Z 355.982,A -85,B 0,C 180,E1 -12962.223,E2 -12962.223} C_VEL
LIN {X 0,Y 362.154,Z 356.001,A -85,B 0,C 180,E1 -12966.686,E2 -12966.686} C_VEL
LIN {X 0,Y 362.036,Z 356.016,A -85,B 0,C 180,E1 -12970.062,E2 -12970.062} C_VEL
LIN {X 0,Y 362.003,Z 356.017,A -85,B 0,C 180,E1 -12973.899,E2 -12973.899} C_VEL
LIN {X 0,Y 361.971,Z 356.025,A -85,B 0,C 180,E1 -12977.938,E2 -12977.938} C_VEL
LIN {X 0,Y 361.896,Z 356.036,A -85,B 0,C 180,E1 -12981.652,E2 -12981.652} C_VEL
LIN {X 0,Y 361.932,Z 356.025,A -85,B 0,C 180,E1 -12985.29,E2 -12985.29} C_VEL
LIN {X 0,Y 361.922,Z 356.028,A -85,B 0,C 180,E1 -12987.778,E2 -12987.778} C_VEL
LIN {X 0,Y 361.85,Z 356.039,A -85,B 0,C 180,E1 -12991.285,E2 -12991.285} C_VEL
LIN {X 0,Y 361.858,Z 356.037,A -85,B 0,C 180,E1 -12994.28,E2 -12994.28} C_VEL
LIN {X 0,Y 361.867,Z 356.038,A -85,B 0,C 180,E1 -12997.223,E2 -12997.223} C_VEL
LIN {X 0,Y 361.854,Z 356.038,A -85,B 0,C 180,E1 -13000.758,E2 -13000.758} C_VEL
LIN {X 0,Y 361.904,Z 356.298,A -85,B 0,C 180,E1 -13001.32,E2 -13001.32} C_VEL
LIN {X 0,Y 363.083,Z 362.018,A -85,B 0,C 180,E1 -13004.951,E2 -13004.951} C_VEL
LIN {X 0,Y 364.132,Z 367.585,A -85,B 0,C 180,E1 -13008.207,E2 -13008.207} C_VEL
LIN {X 0,Y 365.462,Z 374.653,A -85,B 0,C 180,E1 -13012.041,E2 -13012.041} C_VEL
LIN {X 0,Y 365.854,Z 378.092,A -85,B 0,C 180,E1 -13013.786,E2 -13013.786} C_VEL
LIN {X 0,Y 365.243,Z 382.975,A -85,B 0,C 180,E1 -13016.081,E2 -13016.081} C_VEL
LIN {X 0,Y 364.237,Z 389.87,A -85,B 0,C 180,E1 -13019.248,E2 -13019.248} C_VEL
LIN {X 0,Y 363.352,Z 396.46,A -85,B 0,C 180,E1 -13022.243,E2 -13022.243} C_VEL
LIN {X 0,Y 367.959,Z 414.198,A -85,B 0,C 180,E1 -13023.131,E2 -13023.131} C_VEL
LIN {X 0,Y 370.796,Z 428.444,A -85,B 0,C 180,E1 -13023.993,E2 -13023.993} C_VEL
LIN {X 0,Y 372.546,Z 441.232,A -85,B 0,C 180,E1 -13024.892,E2 -13024.892} C_VEL
LIN {X 0,Y 371.177,Z 454.691,A -85,B 0,C 180,E1 -13025.829,E2 -13025.829} C_VEL
LIN {X 0,Y 369.478,Z 468.696,A -85,B 0,C 180,E1 -13027.049,E2 -13027.049} C_VEL
LIN {X 0,Y 367.891,Z 480.253,A -85,B 0,C 180,E1 -13028.276,E2 -13028.276} C_VEL
LIN {X 0,Y 366.231,Z 492.146,A -85,B 0,C 180,E1 -13029.792,E2 -13029.792} C_VEL
LIN {X 0,Y 364.834,Z 503.06,A -85,B 0,C 180,E1 -13031.467,E2 -13031.467} C_VEL
LIN {X 0,Y 363.33,Z 513.69,A -85,B 0,C 180,E1 -13033.422,E2 -13033.422} C_VEL
LIN {X 0,Y 362.3,Z 522.544,A -85,B 0,C 180,E1 -13035.393,E2 -13035.393} C_VEL
LIN {X 0,Y 361.557,Z 528.972,A -85,B 0,C 180,E1 -13037.083,E2 -13037.083} C_VEL
LIN {X 0,Y 360.886,Z 535.991,A -85,B 0,C 180,E1 -13039.338,E2 -13039.338} C_VEL
LIN {X 0,Y 360.557,Z 541.504,A -85,B 0,C 180,E1 -13041.594,E2 -13041.594} C_VEL
LIN {X 0,Y 360.39,Z 545.883,A -85,B 0,C 180,E1 -13044.017,E2 -13044.017} C_VEL
LIN {X 0,Y 360.377,Z 547.82,A -85,B 0,C 180,E1 -13045.526,E2 -13045.526} C_VEL
LIN {X 0,Y 360.378,Z 549.696,A -85,B 0,C 180,E1 -13047.765,E2 -13047.765} C_VEL
LIN {X 0,Y 360.474,Z 550.338,A -85,B 0,C 180,E1 -13050,E2 -13050} C_VEL
LIN {X 0,Y 360.379,Z 549.69,A -85,B 0,C 180,E1 -13052.235,E2 -13052.235} C_VEL
LIN {X 0,Y 360.382,Z 547.806,A -85,B 0,C 180,E1 -13054.474,E2 -13054.474} C_VEL
LIN {X 0,Y 360.477,Z 544.668,A -85,B 0,C 180,E1 -13056.718,E2 -13056.718} C_VEL
LIN {X 0,Y 360.614,Z 540.206,A -85,B 0,C 180,E1 -13058.97,E2 -13058.97} C_VEL
LIN {X 0,Y 361.055,Z 534.325,A -85,B 0,C 180,E1 -13061.224,E2 -13061.224} C_VEL
LIN {X 0,Y 361.671,Z 526.869,A -85,B 0,C 180,E1 -13063.485,E2 -13063.485} C_VEL
LIN {X 0,Y 362.663,Z 518.901,A -85,B 0,C 180,E1 -13065.454,E2 -13065.454} C_VEL
LIN {X 0,Y 363.863,Z 509.322,A -85,B 0,C 180,E1 -13067.421,E2 -13067.421} C_VEL
LIN {X 0,Y 365.217,Z 499.575,A -85,B 0,C 180,E1 -13069.095,E2 -13069.095} C_VEL
LIN {X 0,Y 366.828,Z 488.005,A -85,B 0,C 180,E1 -13070.759,E2 -13070.759} C_VEL
LIN {X 0,Y 368.532,Z 475.273,A -85,B 0,C 180,E1 -13072.273,E2 -13072.273} C_VEL
LIN {X 0,Y 370.151,Z 462.731,A -85,B 0,C 180,E1 -13073.499,E2 -13073.499} C_VEL
LIN {X 0,Y 371.799,Z 449.12,A -85,B 0,C 180,E1 -13074.574,E2 -13074.574} C_VEL
LIN {X 0,Y 372.5,Z 439.69,A -85,B 0,C 180,E1 -13075.203,E2 -13075.203} C_VEL
LIN {X 0,Y 370.148,Z 424.983,A -85,B 0,C 180,E1 -13076.215,E2 -13076.215} C_VEL
LIN {X 0,Y 366.956,Z 410.011,A -85,B 0,C 180,E1 -13077.076,E2 -13077.076} C_VEL
LIN {X 0,Y 363.37,Z 396.469,A -85,B 0,C 180,E1 -13077.736,E2 -13077.736} C_VEL
LIN {X 0,Y 364.654,Z 387.092,A -85,B 0,C 180,E1 -13082.004,E2 -13082.004} C_VEL
LIN {X 0,Y 365.653,Z 380.177,A -85,B 0,C 180,E1 -13085.213,E2 -13085.213} C_VEL
LIN {X 0,Y 365.828,Z 377.376,A -85,B 0,C 180,E1 -13086.552,E2 -13086.552} C_VEL
LIN {X 0,Y 365.188,Z 373.168,A -85,B 0,C 180,E1 -13088.716,E2 -13088.716} C_VEL
LIN {X 0,Y 363.871,Z 366.198,A -85,B 0,C 180,E1 -13092.533,E2 -13092.533} C_VEL
LIN {X 0,Y 362.811,Z 360.759,A -85,B 0,C 180,E1 -13095.785,E2 -13095.785} C_VEL
LIN {X 0,Y 361.866,Z 356.023,A -85,B 0,C 180,E1 -13098.838,E2 -13098.838} C_VEL
LIN {X 0,Y 361.876,Z 356.036,A -85,B 0,C 180,E1 -13101.577,E2 -13101.577} C_VEL
LIN {X 0,Y 361.876,Z 356.039,A -85,B 0,C 180,E1 -13104.655,E2 -13104.655} C_VEL
LIN {X 0,Y 361.839,Z 356.041,A -85,B 0,C 180,E1 -13108.371,E2 -13108.371} C_VEL
LIN {X 0,Y 361.902,Z 356.033,A -85,B 0,C 180,E1 -13110.956,E2 -13110.956} C_VEL
LIN {X 0,Y 361.957,Z 356.025,A -85,B 0,C 180,E1 -13113.475,E2 -13113.475} C_VEL
LIN {X 0,Y 361.893,Z 356.031,A -85,B 0,C 180,E1 -13117.145,E2 -13117.145} C_VEL
LIN {X 0,Y 361.924,Z 356.026,A -85,B 0,C 180,E1 -13120.725,E2 -13120.725} C_VEL
LIN {X 0,Y 361.95,Z 356.019,A -85,B 0,C 180,E1 -13124.226,E2 -13124.226} C_VEL
LIN {X 0,Y 362.003,Z 356.014,A -85,B 0,C 180,E1 -13126.528,E2 -13126.528} C_VEL
LIN {X 0,Y 362.034,Z 356.01,A -85,B 0,C 180,E1 -13129.938,E2 -13129.938} C_VEL
LIN {X 0,Y 362.155,Z 355.994,A -85,B 0,C 180,E1 -13133.314,E2 -13133.314} C_VEL
LIN {X 0,Y 362.284,Z 355.978,A -85,B 0,C 180,E1 -13137.777,E2 -13137.777} C_VEL
LIN {X 0,Y 362.43,Z 355.96,A -85,B 0,C 180,E1 -13140,E2 -13140} C_VEL
LIN {X 0,Y 362.284,Z 355.982,A -85,B 0,C 180,E1 -13142.224,E2 -13142.224} C_VEL
LIN {X 0,Y 362.176,Z 355.995,A -85,B 0,C 180,E1 -13146.686,E2 -13146.686} C_VEL
LIN {X 0,Y 362.079,Z 356.007,A -85,B 0,C 180,E1 -13148.933,E2 -13148.933} C_VEL
LIN {X 0,Y 361.97,Z 356.02,A -85,B 0,C 180,E1 -13152.332,E2 -13152.332} C_VEL
LIN {X 0,Y 361.966,Z 356.019,A -85,B 0,C 180,E1 -13154.62,E2 -13154.62} C_VEL
LIN {X 0,Y 361.963,Z 356.019,A -85,B 0,C 180,E1 -13158.099,E2 -13158.099} C_VEL
LIN {X 0,Y 361.895,Z 356.028,A -85,B 0,C 180,E1 -13161.653,E2 -13161.653} C_VEL
LIN {X 0,Y 361.932,Z 356.028,A -85,B 0,C 180,E1 -13165.29,E2 -13165.29} C_VEL
LIN {X 0,Y 361.922,Z 356.026,A -85,B 0,C 180,E1 -13167.778,E2 -13167.778} C_VEL
LIN {X 0,Y 361.85,Z 356.037,A -85,B 0,C 180,E1 -13171.285,E2 -13171.285} C_VEL
LIN {X 0,Y 361.857,Z 356.036,A -85,B 0,C 180,E1 -13174.28,E2 -13174.28} C_VEL
LIN {X 0,Y 361.866,Z 356.037,A -85,B 0,C 180,E1 -13177.223,E2 -13177.223} C_VEL
LIN {X 0,Y 361.839,Z 356.04,A -85,B 0,C 180,E1 -13180.755,E2 -13180.755} C_VEL
LIN {X 0,Y 361.82,Z 356.043,A -85,B 0,C 180,E1 -13184.368,E2 -13184.368} C_VEL
LIN {X 0,Y 361.865,Z 356.238,A -85,B 0,C 180,E1 -13185.023,E2 -13185.023} C_VEL
LIN {X 0,Y 362.368,Z 358.935,A -85,B 0,C 180,E1 -13187.477,E2 -13187.477} C_VEL
LIN {X 0,Y 362.71,Z 362.164,A -85,B 0,C 180,E1 -13190.251,E2 -13190.251} C_VEL
LIN {X 0,Y 362.709,Z 365.631,A -85,B 0,C 180,E1 -13193.082,E2 -13193.082} C_VEL
LIN {X 0,Y 362.368,Z 370.026,A -85,B 0,C 180,E1 -13196.509,E2 -13196.509} C_VEL
LIN {X 0,Y 362.014,Z 374.286,A -85,B 0,C 180,E1 -13199.685,E2 -13199.685} C_VEL
LIN {X 0,Y 361.722,Z 379.575,A -85,B 0,C 180,E1 -13203.457,E2 -13203.457} C_VEL
LIN {X 0,Y 361.601,Z 381.617,A -85,B 0,C 180,E1 -13204.864,E2 -13204.864} C_VEL
LIN {X 0,Y 367.045,Z 397.923,A -85,B 0,C 180,E1 -13205.802,E2 -13205.802} C_VEL
LIN {X 0,Y 370.606,Z 411.131,A -85,B 0,C 180,E1 -13206.697,E2 -13206.697} C_VEL
LIN {X 0,Y 372.617,Z 420.304,A -85,B 0,C 180,E1 -13207.402,E2 -13207.402} C_VEL
LIN {X 0,Y 371.473,Z 434.36,A -85,B 0,C 180,E1 -13208.411,E2 -13208.411} C_VEL
LIN {X 0,Y 370.164,Z 445.789,A -85,B 0,C 180,E1 -13209.437,E2 -13209.437} C_VEL
LIN {X 0,Y 368.493,Z 458.005,A -85,B 0,C 180,E1 -13210.792,E2 -13210.792} C_VEL
LIN {X 0,Y 367.154,Z 468.069,A -85,B 0,C 180,E1 -13212.165,E2 -13212.165} C_VEL
LIN {X 0,Y 365.575,Z 478.068,A -85,B 0,C 180,E1 -13213.815,E2 -13213.815} C_VEL
LIN {X 0,Y 364.373,Z 486.352,A -85,B 0,C 180,E1 -13215.478,E2 -13215.478} C_VEL
LIN {X 0,Y 363.118,Z 494.267,A -85,B 0,C 180,E1 -13217.424,E2 -13217.424} C_VEL
LIN {X 0,Y 362.165,Z 500.657,A -85,B 0,C 180,E1 -13219.377,E2 -13219.377} C_VEL
LIN {X 0,Y 361.378,Z 506.332,A -85,B 0,C 180,E1 -13221.613,E2 -13221.613} C_VEL
LIN {X 0,Y 361.029,Z 509.61,A -85,B 0,C 180,E1 -13223.293,E2 -13223.293} C_VEL
LIN {X 0,Y 360.632,Z 512.758,A -85,B 0,C 180,E1 -13225.529,E2 -13225.529} C_VEL
LIN {X 0,Y 360.588,Z 514.605,A -85,B 0,C 180,E1 -13227.766,E2 -13227.766} C_VEL
LIN {X 0,Y 360.477,Z 515.236,A -85,B 0,C 180,E1 -13230,E2 -13230} C_VEL
LIN {X 0,Y 360.587,Z 514.661,A -85,B 0,C 180,E1 -13232.234,E2 -13232.234} C_VEL
LIN {X 0,Y 360.63,Z 512.874,A -85,B 0,C 180,E1 -13234.471,E2 -13234.471} C_VEL
LIN {X 0,Y 361.029,Z 509.788,A -85,B 0,C 180,E1 -13236.708,E2 -13236.708} C_VEL
LIN {X 0,Y 361.52,Z 505.307,A -85,B 0,C 180,E1 -13238.947,E2 -13238.947} C_VEL
LIN {X 0,Y 362.357,Z 499.27,A -85,B 0,C 180,E1 -13241.184,E2 -13241.184} C_VEL
LIN {X 0,Y 363.383,Z 492.542,A -85,B 0,C 180,E1 -13243.135,E2 -13243.135} C_VEL
LIN {X 0,Y 364.745,Z 484.316,A -85,B 0,C 180,E1 -13245.051,E2 -13245.051} C_VEL
LIN {X 0,Y 365.965,Z 475.483,A -85,B 0,C 180,E1 -13246.742,E2 -13246.742} C_VEL
LIN {X 0,Y 367.602,Z 464.905,A -85,B 0,C 180,E1 -13248.389,E2 -13248.389} C_VEL
LIN {X 0,Y 369.12,Z 454.203,A -85,B 0,C 180,E1 -13249.753,E2 -13249.753} C_VEL
LIN {X 0,Y 370.559,Z 442.502,A -85,B 0,C 180,E1 -13250.977,E2 -13250.977} C_VEL
LIN {X 0,Y 371.865,Z 430.479,A -85,B 0,C 180,E1 -13251.99,E2 -13251.99} C_VEL
LIN {X 0,Y 372.707,Z 421.05,A -85,B 0,C 180,E1 -13252.646,E2 -13252.646} C_VEL
LIN {X 0,Y 370.019,Z 408.643,A -85,B 0,C 180,E1 -13253.588,E2 -13253.588} C_VEL
LIN {X 0,Y 366.097,Z 394.826,A -85,B 0,C 180,E1 -13254.498,E2 -13254.498} C_VEL
LIN {X 0,Y 361.703,Z 382.15,A -85,B 0,C 180,E1 -13255.207,E2 -13255.207} C_VEL
LIN {X 0,Y 361.615,Z 381.571,A -85,B 0,C 180,E1 -13255.269,E2 -13255.269} C_VEL
LIN {X 0,Y 361.721,Z 379.732,A -85,B 0,C 180,E1 -13256.535,E2 -13256.535} C_VEL
LIN {X 0,Y 361.166,Z 378.52,A -85,B 0,C 180,E1 -13257.446,E2 -13257.446} C_VEL
LIN {X 0,Y 358.424,Z 376.861,A -85,B 0,C 180,E1 -13258.94,E2 -13258.94} C_VEL
LIN {X 0,Y 356.095,Z 375.587,A -85,B 0,C 180,E1 -13260.152,E2 -13260.152} C_VEL
LIN {X 0,Y 355.157,Z 374.501,A -85,B 0,C 180,E1 -13261.084,E2 -13261.084} C_VEL
LIN {X 0,Y 355.117,Z 374.097,A -85,B 0,C 180,E1 -13261.397,E2 -13261.397} C_VEL
LIN {X 0,Y 355.48,Z 369.416,A -85,B 0,C 180,E1 -13264.984,E2 -13264.984} C_VEL
LIN {X 0,Y 355.773,Z 365.926,A -85,B 0,C 180,E1 -13267.798,E2 -13267.798} C_VEL
LIN {X 0,Y 355.659,Z 362.504,A -85,B 0,C 180,E1 -13270.7,E2 -13270.7} C_VEL
LIN {X 0,Y 355.162,Z 358.95,A -85,B 0,C 180,E1 -13273.836,E2 -13273.836} C_VEL
LIN {X 0,Y 354.797,Z 356.914,A -85,B 0,C 180,E1 -13275.792,E2 -13275.792} C_VEL
LIN {X 0,Y 354.792,Z 356.912,A -85,B 0,C 180,E1 -13279.179,E2 -13279.179} C_VEL
LIN {X 0,Y 354.811,Z 356.911,A -85,B 0,C 180,E1 -13282.403,E2 -13282.403} C_VEL
LIN {X 0,Y 354.816,Z 356.915,A -85,B 0,C 180,E1 -13284.941,E2 -13284.941} C_VEL
LIN {X 0,Y 354.798,Z 356.918,A -85,B 0,C 180,E1 -13288.405,E2 -13288.405} C_VEL
LIN {X 0,Y 354.855,Z 356.907,A -85,B 0,C 180,E1 -13291.619,E2 -13291.619} C_VEL
LIN {X 0,Y 354.904,Z 356.898,A -85,B 0,C 180,E1 -13294.173,E2 -13294.173} C_VEL
LIN {X 0,Y 354.84,Z 356.911,A -85,B 0,C 180,E1 -13297.894,E2 -13297.894} C_VEL
LIN {X 0,Y 354.927,Z 356.896,A -85,B 0,C 180,E1 -13301.892,E2 -13301.892} C_VEL
LIN {X 0,Y 354.948,Z 356.895,A -85,B 0,C 180,E1 -13305.981,E2 -13305.981} C_VEL
LIN {X 0,Y 354.983,Z 356.893,A -85,B 0,C 180,E1 -13309.736,E2 -13309.736} C_VEL
LIN {X 0,Y 355.12,Z 356.873,A -85,B 0,C 180,E1 -13312.037,E2 -13312.037} C_VEL
LIN {X 0,Y 355.098,Z 356.875,A -85,B 0,C 180,E1 -13314.321,E2 -13314.321} C_VEL
LIN {X 0,Y 355.249,Z 356.856,A -85,B 0,C 180,E1 -13317.732,E2 -13317.732} C_VEL
LIN {X 0,Y 355.401,Z 356.842,A -85,B 0,C 180,E1 -13320,E2 -13320} C_VEL
LIN {X 0,Y 355.249,Z 356.858,A -85,B 0,C 180,E1 -13322.267,E2 -13322.267} C_VEL
LIN {X 0,Y 355.117,Z 356.877,A -85,B 0,C 180,E1 -13326.819,E2 -13326.819} C_VEL
LIN {X 0,Y 354.984,Z 356.892,A -85,B 0,C 180,E1 -13330.264,E2 -13330.264} C_VEL
LIN {X 0,Y 354.948,Z 356.896,A -85,B 0,C 180,E1 -13334.019,E2 -13334.019} C_VEL
LIN {X 0,Y 354.927,Z 356.903,A -85,B 0,C 180,E1 -13338.108,E2 -13338.108} C_VEL
LIN {X 0,Y 354.839,Z 356.911,A -85,B 0,C 180,E1 -13342.106,E2 -13342.106} C_VEL
LIN {X 0,Y 354.903,Z 356.903,A -85,B 0,C 180,E1 -13345.827,E2 -13345.827} C_VEL
LIN {X 0,Y 354.857,Z 356.906,A -85,B 0,C 180,E1 -13349.678,E2 -13349.678} C_VEL
LIN {X 0,Y 354.809,Z 356.917,A -85,B 0,C 180,E1 -13353.702,E2 -13353.702} C_VEL
LIN {X 0,Y 354.802,Z 356.919,A -85,B 0,C 180,E1 -13356.459,E2 -13356.459} C_VEL
LIN {X 0,Y 354.826,Z 356.914,A -85,B 0,C 180,E1 -13360.441,E2 -13360.441} C_VEL
LIN {X 0,Y 355.836,Z 361.839,A -85,B 0,C 180,E1 -13363.731,E2 -13363.731} C_VEL
LIN {X 0,Y 356.975,Z 367.83,A -85,B 0,C 180,E1 -13367.394,E2 -13367.394} C_VEL
LIN {X 0,Y 358.229,Z 374.446,A -85,B 0,C 180,E1 -13371.112,E2 -13371.112} C_VEL
LIN {X 0,Y 358.886,Z 378.788,A -85,B 0,C 180,E1 -13373.407,E2 -13373.407} C_VEL
LIN {X 0,Y 358.474,Z 382.937,A -85,B 0,C 180,E1 -13375.429,E2 -13375.429} C_VEL
LIN {X 0,Y 357.212,Z 391.02,A -85,B 0,C 180,E1 -13379.233,E2 -13379.233} C_VEL
LIN {X 0,Y 356.453,Z 396.285,A -85,B 0,C 180,E1 -13381.698,E2 -13381.698} C_VEL
LIN {X 0,Y 360.941,Z 413.436,A -85,B 0,C 180,E1 -13382.576,E2 -13382.576} C_VEL
LIN {X 0,Y 363.871,Z 427.643,A -85,B 0,C 180,E1 -13383.46,E2 -13383.46} C_VEL
LIN {X 0,Y 365.967,Z 441.959,A -85,B 0,C 180,E1 -13384.499,E2 -13384.499} C_VEL
LIN {X 0,Y 364.456,Z 455.913,A -85,B 0,C 180,E1 -13385.506,E2 -13385.506} C_VEL
LIN {X 0,Y 362.703,Z 469.641,A -85,B 0,C 180,E1 -13386.746,E2 -13386.746} C_VEL
LIN {X 0,Y 360.947,Z 482.17,A -85,B 0,C 180,E1 -13388.137,E2 -13388.137} C_VEL
LIN {X 0,Y 359.294,Z 493.179,A -85,B 0,C 180,E1 -13389.604,E2 -13389.604} C_VEL
LIN {X 0,Y 357.782,Z 504.315,A -85,B 0,C 180,E1 -13391.385,E2 -13391.385} C_VEL
